# B&R Automation Studio project Panasonic_LinkaPowerCP2_A2021055 (part 7)

#### MaticaSet.st
```iecst
(* Skrutkovací set maticovačky *)
FUNCTION_BLOCK MaticaSet

	//Príznak matica pripravena//
	STAV.MaticaPripravena:= IN.PritomnostMaticeNaVystupe AND IN.PodavacMatice_ZASUNUTY;

	//*******************************Ovládanie zhadzovacieho vzduchu pred lištou zásobníka******************************************//
	Internal.CasZaplneniaZasobnika.IN:= IN.ZaplnenieListyZasobnika AND OUT.VibropohonZasobnika_RUN;

	IF Internal.CasZaplneniaZasobnika.Q THEN
		OUT.ZhadzovaciVzduch_RUN:= TRUE;
	ELSE
		OUT.ZhadzovaciVzduch_RUN:= FALSE;
	END_IF

	Internal.CasZaplneniaZasobnika.PT:= T#1s;
	Internal.CasZaplneniaZasobnika();

	//******************************Vypnutie triediaceho vzduchu nad lištou zásobníka************************************************//
	Internal.CasVypnTriediacehoVzduchu.IN:= OUT.TriediaciVzduch_RUN AND NOT OUT.VibropohonZasobnika_RUN;
	IF Internal.CasVypnTriediacehoVzduchu.Q THEN
		OUT.TriediaciVzduch_RUN:= FALSE;
	END_IF

	Internal.CasVypnTriediacehoVzduchu.PT:= T#1s;
	Internal.CasVypnTriediacehoVzduchu();

	//*******************************Vypnutie zásobníka***************************************//
	Internal.CasVypnZasobnika.IN:= IN.ZaplnenieListyZasobnika AND OUT.VibropohonZasobnika_RUN;

	IF Internal.CasVypnZasobnika.Q THEN
		OUT.VibropohonZasobnika_RUN:= FALSE;
	END_IF

	Internal.CasVypnZasobnika.PT:= T#3s;
	Internal.CasVypnZasobnika();

	//*******************************Zapnutie zásobníka keď je prázdna lišta zásobníka*****************//
	IF CMD.ENABLE AND NOT STAV.ERROR AND NOT IN.ZaplnenieListyZasobnika AND NOT OUT.VibropohonZasobnika_RUN AND IN.PodavacMatice_ZASUNUTY THEN
		OUT.VibropohonZasobnika_RUN:= TRUE;
	END_IF

	//***********************************Enable knižnice***************************************//
	IF NOT CMD.ENABLE AND Step <> 0 THEN
		OUT.VibropohonZasobnika_RUN:= FALSE;
		OUT.ZhadzovaciVzduch_RUN:= FALSE;
		OUT.NastrelenieMatice_RUN:= FALSE;
		Internal.PoInit:= FALSE;
		STAV.ERROR:= FALSE;
		STAV.PodanieMatice_BUSY:= FALSE;
		STAV.CisloPoruchy:= 0;
		STAV.PopisPoruchy:= '';
		Step:= 0;
	END_IF

	//**********************************Reset poruchy*****************************************//
	//1 - porucha preletu matice cez snímač za oddelovačom
	//2 - porucha preletu matice cez snimač pred podavačom
	//3 - porucha otočenia oddelovača smerom k zásobníku
	//4 - porucha otočenia oddelovača smerom k maticovačke
	//5 - porucha vysunutia podavača vpred
	//6 - porucha zasunutia podavača vzad
	//7 - porucha snimača prítomnosti matice v skrutkovačke

	IF CMD.ResetPoruchy THEN
		STAV.ERROR:= FALSE;
		STAV.CisloPoruchy:= 0;
		STAV.PopisPoruchy:= '';
	END_IF

	CASE Step OF

		0: //Nulovanie//
			Internal.IdleTime_200ms.IN:= FALSE;
			Internal.IdleTime_100ms.IN:= FALSE;
			Internal.IdleTime_500ms.IN:= FALSE;
			Internal.IdleTime_1s.IN:= FALSE;
			Internal.IdleTime_1500ms.IN:= FALSE;
			Internal.AlarmTime_3s.IN:= FALSE;
			OUT.PodavacMatice_Vysun:= FALSE;
			OUT.OtocOddelovacMatice_NaVystup:= FALSE;
			OUT.NastrelenieMatice_RUN:= FALSE;
			CMD.RR_OtocPodavac_Vstup:= FALSE;
			CMD.RR_OtocPodavac_Vystup:= FALSE;
			CMD.RR_VysunPodavacMatic:= FALSE;
			CMD.RR_ZapniZasobnik:= FALSE;
			CMD.RucnyRezim:= FALSE;
			CMD.PodajMaticu:=FALSE;
			STAV.PodanieMatice_BUSY:= FALSE;
			IF NOT CMD.PodajMaticu AND CMD.ENABLE AND NOT STAV.ERROR THEN
				Step:= 1;
			END_IF

		1: //Čakam na spustenie//
			IF CMD.RucnyRezim THEN
				Step:= 70;
			ELSIF CMD.PodajMaticu THEN
				Step:= 10;
			END_IF

		10: //Kontrola matice na vystupe//
			STAV.PodanieMatice_BUSY:= TRUE;
			IF IN.PritomnostMaticeNaVystupe THEN
				Step:= 0;
			ELSE
				IF NOT Internal.PoInit THEN
					Step:= 11;
				ELSE
					Step:= 13;
				END_IF
			END_IF

		11: //Hladanie matice pri prvom spusteni//
			OUT.PodavacMatice_Vysun:= FALSE;
			Internal.IdleTime_1500ms.IN:= OUT.NastrelenieMatice_RUN;

			IF IN.PodavacMatice_ZASUNUTY THEN
				OUT.NastrelenieMatice_RUN:= TRUE;
			END_IF

			IF Internal.IdleTime_1500ms.Q THEN
				OUT.NastrelenieMatice_RUN:= FALSE;
				Internal.IdleTime_1500ms.IN:= FALSE;
				Step:= 12;
			END_IF

		12: //Vysunutie podavača//
			OUT.PodavacMatice_Vysun:= TRUE;
			Internal.AlarmTime_3s.IN:= TRUE;
			Internal.IdleTime_500ms.IN:= IN.PodavacMatice_VYSUNUTY;

			IF Internal.IdleTime_500ms.Q THEN
				Internal.PoInit:= TRUE;
				Internal.IdleTime_500ms.IN:= FALSE;
				OUT.PodavacMatice_Vysun:= FALSE;
				Internal.AlarmTime_3s.IN:= FALSE;
				Step:= 10;
			ELSIF Internal.AlarmTime_3s.Q THEN
				STAV.ERROR:= TRUE;
				STAV.CisloPoruchy:= 5;
				STAV.PopisPoruchy:= 'Porucha vysunutia podavača vpred';
				Step:= 0;
			END_IF

		13: //Zasunutie podavaca matice a otocenie oddelovaca k zasobniku//
			OUT.PodavacMatice_Vysun:= FALSE;
			OUT.OtocOddelovacMatice_NaVystup:= FALSE;
			Internal.AlarmTime_3s.IN:= TRUE;

			IF IN.PodavacMatice_ZASUNUTY AND IN.OddelovacOtoceny_VSTUP THEN
				Internal.AlarmTime_3s.IN:= FALSE;
				Step:= 15;
			ELSIF Internal.AlarmTime_3s.Q THEN
				STAV.ERROR:= TRUE;
				IF NOT IN.PodavacMatice_ZASUNUTY THEN
					STAV.CisloPoruchy:= 6;
					STAV.PopisPoruchy:= 'Porucha zasunutia podavača vzad';
				ELSIF NOT IN.OddelovacOtoceny_VSTUP THEN
					STAV.CisloPoruchy:= 3;
					STAV.PopisPoruchy:= 'Porucha otocenia oddelovaca smerom k zasobníku';
				END_IF
				Step:= 0;
			END_IF

		15: //Spustenie zasobnika//
			OUT.TriediaciVzduch_RUN:= TRUE;
			Internal.IdleTime_1s.IN:= OUT.TriediaciVzduch_RUN;
			Internal.IdleTime_1500ms.IN:= IN.ZaplnenieListyZasobnika AND OUT.VibropohonZasobnika_RUN;

			IF Internal.IdleTime_1s.Q THEN
				OUT.VibropohonZasobnika_RUN:= TRUE;
			END_IF

			IF Internal.IdleTime_1500ms.Q THEN
				Internal.IdleTime_1s.IN:= FALSE;
				Internal.IdleTime_1500ms.IN:= FALSE;
				Step:= 18;
			END_IF

		18: //Otočenie oddelovača matic na vystup smerom k maticovačke a čakanie na prechod matice cez prvy snimac//
			OUT.OtocOddelovacMatice_NaVystup:= TRUE;
			Internal.AlarmTime_3s.IN:= TRUE;

			IF IN.Oddelovac_SnimPrechoduMatice THEN
				Internal.AlarmTime_3s.IN:= FALSE;
				Step:= 20;
			ELSIF Internal.AlarmTime_3s.Q THEN
				STAV.ERROR:= TRUE;
				STAV.CisloPoruchy:= 1;
				STAV.PopisPoruchy:= 'Porucha preletu matice cez snimac za oddelovacom';
				Step:= 0;
			END_IF

		20: //Zapnutie nastrelovacieho vzduchu a čakanie na prechod matice cez druhý snímač//
			OUT.NastrelenieMatice_RUN:= TRUE;
			Internal.AlarmTime_3s.IN:= TRUE;

			IF IN.Podavac_SnimPrechoduMatice THEN
				Internal.AlarmTime_3s.IN:= FALSE;
				Step:= 23;
			ELSIF Internal.AlarmTime_3s.Q THEN
				STAV.ERROR:= TRUE;
				STAV.CisloPoruchy:= 2;
				STAV.PopisPoruchy:= 'Porucha preletu matice cez snimac pred podavacom';
				Step:= 0;
			END_IF

		23: //Cakam na vysunutie podavaca//
			Internal.IdleTime_500ms.IN:= TRUE;

			IF Internal.IdleTime_500ms.Q THEN
				OUT.PodavacMatice_Vysun:= TRUE;
				Internal.AlarmTime_3s.IN:= TRUE;
			END_IF

			IF IN.PodavacMatice_VYSUNUTY AND IN.PritomnostMaticeNaVystupe THEN
				Internal.IdleTime_500ms.IN:= FALSE;
				Internal.AlarmTime_3s.IN:= FALSE;
				Step:= 25;
			ELSIF Internal.AlarmTime_3s.Q THEN
				STAV.ERROR:= TRUE;
				IF NOT IN.PodavacMatice_VYSUNUTY THEN
					STAV.CisloPoruchy:= 5;
					STAV.PopisPoruchy:= 'Porucha vysunutia podavaca vpred';
				ELSIF NOT IN.PritomnostMaticeNaVystupe THEN
					STAV.CisloPoruchy:= 7;
					STAV.PopisPoruchy:= 'Porucha snimaca pritomnosti matice v skrutkovacke';
				END_IF
				Step:= 0;
			END_IF

		25: //Čakam na zasunutie podavača//
			Internal.IdleTime_200ms.IN:= TRUE;

			IF Internal.IdleTime_200ms.Q THEN
				OUT.PodavacMatice_Vysun:= FALSE;
				Internal.AlarmTime_3s.IN:= TRUE;
			END_IF

			IF IN.PodavacMatice_ZASUNUTY THEN
				Internal.IdleTime_200ms.IN:= FALSE;
				Internal.AlarmTime_3s.IN:= FALSE;
				Step:= 0;
			ELSIF Internal.AlarmTime_3s.Q THEN
				STAV.ERROR:= TRUE;
				STAV.CisloPoruchy:= 6;
				STAV.PopisPoruchy:= 'Porucha zasunutia podavaca vzad';
				Step:= 0;
			END_IF

		70: //Rucny rezim//
			IF CMD.RR_ZapniZasobnik THEN
				OUT.TriediaciVzduch_RUN:= TRUE;
				Internal.IdleTime_1s.IN:= TRUE;
			ELSE
				Internal.IdleTime_1s.IN:= FALSE;
			END_IF

			OUT.VibropohonZasobnika_RUN:= Internal.IdleTime_1s.Q;

			IF NOT CMD.RucnyRezim THEN
				OUT.VibropohonZasobnika_RUN:= FALSE;
				Step:= 0;
			ELSIF CMD.PodajMaticu THEN
				OUT.PodavacMatice_Vysun:= FALSE;
				Step:= 10;
			END_IF

			IF CMD.RR_OtocPodavac_Vstup THEN
				OUT.OtocOddelovacMatice_NaVystup:= FALSE;
				CMD.RR_OtocPodavac_Vstup:= FALSE;
			ELSIF CMD.RR_OtocPodavac_Vystup THEN
				OUT.OtocOddelovacMatice_NaVystup:= TRUE;
				CMD.RR_OtocPodavac_Vystup:= FALSE;
			END_IF

			OUT.PodavacMatice_Vysun:= CMD.RR_VysunPodavacMatic;

	END_CASE

	//*****************Časovače************************//
	Internal.IdleTime_100ms.PT:= T#200ms;
	Internal.IdleTime_100ms();
	Internal.IdleTime_200ms.PT:= T#200ms;
	Internal.IdleTime_200ms();
	Internal.IdleTime_500ms.PT:= T#200ms;
	Internal.IdleTime_500ms();
	Internal.IdleTime_1s.PT:= T#1s;
	Internal.IdleTime_1s();
	Internal.IdleTime_1500ms.PT:= T#1s500ms;
	Internal.IdleTime_1500ms();
	Internal.AlarmTime_3s.PT:= T#40s;
	Internal.AlarmTime_3s();

END_FUNCTION_BLOCK
```

### Library Logical/Libraries/RoCa_Festo (IEC, version 1.00.0)

#### Types.typ - Exported data types
```iecst
TYPE
	OutputRawStruc : 	STRUCT
		Control_word_or_setpoint_0 : UINT;
		Control_word_or_setpoint_1 : UINT;
		Control_word_or_setpoint_2 : UINT;
		Control_word_or_setpoint_3 : UINT;
		Control_word_or_setpoint_4 : UINT;
		Control_word_or_setpoint_5 : UINT;
		Control_word_or_setpoint_6 : UINT;
		Control_word_or_setpoint_7 : UINT;
		Control_word_or_setpoint_8 : UINT;
		Control_word_or_setpoint_9 : UINT;
		Control_word_or_setpoint_10 : UINT;
		Control_word_or_setpoint_11 : UINT;
		Control_word_or_setpoint_12 : UINT;
		Control_word_or_setpoint_13 : UINT;
		Control_word_or_setpoint_14 : UINT;
		Control_word_or_setpoint_15 : UINT;
		User1 : UINT;
		MDI_decceleration : UINT;
		MDI_acceleration : UINT;
		MDI_velocity : UDINT;
		MDI_target_position : UDINT;
		Override : UINT;
		Position_Controlword_2 : UINT;
		Position_Controlword_1 : UINT;
		Control_word_2 : UINT;
		Control_word_1 : UINT;
	END_STRUCT;
	InputRawStruc : 	STRUCT
		Status_word_or_actual_value_0 : UINT;
		Status_word_or_actual_value_1 : UINT;
		Status_word_or_actual_value_2 : UINT;
		Status_word_or_actual_value_3 : UINT;
		Status_word_or_actual_value_4 : UINT;
		Status_word_or_actual_value_5 : UINT;
		Status_word_or_actual_value_6 : UINT;
		Status_word_or_actual_value_7 : UINT;
		Status_word_or_actual_value_8 : UINT;
		Status_word_or_actual_value_9 : UINT;
		Status_word_or_actual_value_10 : UINT;
		Status_word_or_actual_value_11 : UINT;
		Status_word_or_actual_value_12 : UINT;
		Status_word_or_actual_value_13 : UINT;
		Status_word_or_actual_value_14 : UINT;
		Status_word_or_actual_value_15 : UINT;
		User : UINT;
		Warn_Code : UINT;
		Fault_Code : UINT;
		Speed_actual_value_B : UDINT;
		Position_actual_value_A : UDINT;
		Report_word : UINT;
		Position_Statusword_2 : UINT;
		Position_Statusword_1 : UINT;
		Status_word_2 : UINT;
		Status_word_1 : UINT;
	END_STRUCT;
	OutputStruc : 	STRUCT
		ExtendedParam0 : UINT;
		ExtendedParam1 : UINT;
		ExtendedParam2 : UINT;
		ExtendedParam3 : UINT;
		ExtendedParam4 : UINT;
		ExtendedParam5 : UINT;
		ExtendedParam6 : UINT;
		ExtendedParam7 : UINT;
		ExtendedParam8 : UINT;
		ExtendedParam9 : UINT;
		ExtendedParam10 : UINT;
		ExtendedParam11 : UINT;
		ExtendedParam12 : UINT;
		ExtendedParam13 : UINT;
		ExtendedParam14 : UINT;
		ExtendedParam15 : UINT;
		user : UINT;
		TraverseToFixedEndstop_Bit8 : BOOL;
		ActivateHardwLimitSwitch_Bit15 : BOOL;
		ActivateSoftLimitSwitch_Bit14 : BOOL;
		TouchProbeEdgeSelection_Bit11 : BOOL;
		TouchProbeSelection_Bit10 : BOOL;
		JoggingIncremental_Bit5 : BOOL;
		MDIselection_Bit15 : BOOL;
		NegModuloPositioningDir_Bit10 : BOOL;
		PosModuloPositioningDir_Bit9 : BOOL;
		AbsolutePositioning_Bit8 : BOOL;
		TraversingBlockSelection_Bit0 : BOOL;
		TraversingBlockSelection_Bit1 : BOOL;
		TraversingBlockSelection_Bit2 : BOOL;
		TraversingBlockSelection_Bit3 : BOOL;
		TraversingBlockSelection_Bit4 : BOOL;
		TraversingBlockSelection_Bit5 : BOOL;
		TraversingBlockSelection_Bit6 : BOOL;
		OpenHoldingBrake_Bit12 : BOOL;
		StartHomingProcedure_Bit11 : BOOL;
		ControlByPLC_Bit10 : BOOL;
		Jog2_Bit9 : BOOL;
		Jog1_Bit8 : BOOL;
		FaultAck_Bit7 : BOOL;
		ActivateTraversingTask_Bit6 : BOOL;
		NoIntermediateStop_Bit5 : BOOL;
		DoNotRejectTraversingTask_Bit4 : BOOL;
		EnableOperation_Bit3 : BOOL;
		NoQuickStop_Bit2 : BOOL;
		NoCoastStop_Bit1 : BOOL;
		SwitchON_Bit0 : BOOL;
	END_STRUCT;
	InputStruc : 	STRUCT
		ExtendedParam0 : UINT;
		ExtendedParam1 : UINT;
		ExtendedParam2 : UINT;
		ExtendedParam3 : UINT;
		ExtendedParam4 : UINT;
		ExtendedParam5 : UINT;
		ExtendedParam6 : UINT;
		ExtendedParam7 : UINT;
		ExtendedParam8 : UINT;
		ExtendedParam9 : UINT;
		ExtendedParam10 : UINT;
		ExtendedParam11 : UINT;
		ExtendedParam12 : UINT;
		ExtendedParam13 : UINT;
		ExtendedParam14 : UINT;
		ExtendedParam15 : UINT;
		User : UINT;
		WarnCode : UINT;
		FaultCode : UINT;
		Speed : UDINT;
		Position : UDINT;
		PulsesEnabledMELDW_Bit13 : BOOL;
		DriveReady_Bit12 : BOOL;
		ControlerEnabled_Bit11 : BOOL;
		SpeedSetpointDeviationInTol_Bit8 : BOOL;
		PsTempWarningInactive_Bit7 : BOOL;
		MotorTempWarningInactive_Bit6 : BOOL;
		VariableSignalingFunction_Bit5 : BOOL;
		RPMequalThreshold_Bit3 : BOOL;
		RPMlowerThreshold_Bit2 : BOOL;
		TorqUtilLessTorqThres_Bit1 : BOOL;
		RampFunctionCompleted_Bit0 : BOOL;
		PulsesEnabled_Bit11 : BOOL;
		MoveToFixedStopActiveZSW2_Bit8 : BOOL;
		TraversingCommandActive_Bit15 : BOOL;
		MoveToFixedStopActive_Bit14 : BOOL;
		FixedStopClampTorqReached_Bit13 : BOOL;
		FixedStopReached_Bit12 : BOOL;
		DirectOut2ViaTraversBlock_Bit11 : BOOL;
		DirectOut1ViaTraversBlock_Bit10 : BOOL;
		PosActValueLessCamSwitch1_Bit9 : BOOL;
		PosActValueLessCamSwitch0_Bit8 : BOOL;
		SoftwareLimitSwitchPlus_Bit7 : BOOL;
		SoftwareLimitSwitchMinus_Bit6 : BOOL;
		DriveMovesBackwards_Bit5 : BOOL;
		DriveMovesForward_Bit4 : BOOL;
		SetpointAvailable_Bit2 : BOOL;
		VelocityLimitingActive_Bit1 : BOOL;
		TrackingModeActive_Bit0 : BOOL;
		MDIactive_Bit15 : BOOL;
		TraversingBlockActive_Bit13 : BOOL;
		RefPointAproachActive_Bit11 : BOOL;
		JoggingActive_Bit10 : BOOL;
		PositiveLimitSwitch_Bit9 : BOOL;
		NegativeLimitSwitch_Bit8 : BOOL;
		ActiveTravesringBlock_Bit0 : BOOL;
		ActiveTravesringBlock_Bit1 : BOOL;
		ActiveTravesringBlock_Bit2 : BOOL;
		ActiveTravesringBlock_Bit3 : BOOL;
		ActiveTravesringBlock_Bit4 : BOOL;
		ActiveTravesringBlock_Bit5 : BOOL;
		ActiveTravesringBlock_Bit6 : BOOL;
		AxisDeccelerated_Bit15 : BOOL;
		AxisAccelerated_Bit14 : BOOL;
		DriveStopped_Bit13 : BOOL;
		TraversingTaskAck_Bit12 : BOOL;
		HomePositionSet_Bit11 : BOOL;
		TargetPositionReached_Bit10 : BOOL;
		ControlRequested_Bit9 : BOOL;
		FolowingErrorWithinTol_Bit8 : BOOL;
		WarningPresent_Bit7 : BOOL;
		SwitchingOnInhibited_Bit6 : BOOL;
		QuickStopNotActivated_Bit5 : BOOL;
		CoastStopNotActivated_Bit4 : BOOL;
		FaultPresent_Bit3 : BOOL;
		OperationEnabled_Bit2 : BOOL;
		ReadyToOperate_Bit1 : BOOL;
		ReadyToSwitchON_Bit0 : BOOL;
	END_STRUCT;
	FestoServoDriverStruc : 	STRUCT
		OUT_forMapping : OutputRawStruc;
		IN_forMapping : InputRawStruc;
		OUT : OutputStruc;
		IN : InputStruc;
		Step : USINT;
		Info : WSTRING[80];
		Status : StatusStruc;
		Command : CommandStruc;
		Parameters : ParamStruc;
	END_STRUCT;
	ParamStruc : 	STRUCT
		Torque : REAL; (*Nm*)
		Distance : REAL; (*vzdialenost pre move additive [mm]*)
		Position : REAL; (*pozicia pre move position [mm]*)
		Override : REAL; (*0-200%*)
		Velocity : REAL; (*m/s*)
		Dcc : REAL; (*m/s2*)
		Acc : REAL; (*m/s2*)
		Jog : JogStruc;
	END_STRUCT;
	CommandStruc : 	STRUCT
		PowerON : BOOL;
		ErrReset : BOOL;
		JogNeg : BOOL;
		JogPos : BOOL;
		MoveAdditive : BOOL;
		MovePosition : BOOL;
		TorqueLimitation : BOOL; (*1-orezava moment na nastaveny v parametroch*)
		Stop : BOOL;
		Pause : BOOL;
	END_STRUCT;
	StatusStruc : 	STRUCT
		WarningMessage : WSTRING[80];
		ErrorMessage : WSTRING[80];
		InTorque : BOOL;
		InPosition : BOOL;
		StandStill : BOOL;
		Warning : BOOL;
		Error : BOOL;
		Ready : BOOL;
		ActTorque : REAL; (*Nm*)
		ActVelocity : REAL; (*mm/s*)
		ActPosition : REAL; (*mm*)
	END_STRUCT;
	JogStruc : 	STRUCT
		Acc : REAL;
		Velocity : REAL;
	END_STRUCT;
	LinearScaling_InternalStruc : 	STRUCT
		ScaleFactor : REAL;
		Offset : REAL;
	END_STRUCT;
	LinearScaling_SettingStruc : 	STRUCT
		InputLowerLimit : REAL; (*Minimum ktore vie vstup dosiahnut*)
		InputUpperLimit : REAL; (*Maximum ktore vie vstup dosiahnut*)
		OutputLowerLimit : REAL; (*Minimum ktore ma vystup ukazovat*)
		OutputUpperLimit : REAL; (*Maximum ktore ma vystup ukazovat*)
	END_STRUCT;
END_TYPE
```

#### RoCa_Festo.fun - Exported functions and function blocks
```iecst
{REDUND_OK} FUNCTION_BLOCK ServoDriver (*Riadenie festo driverov*) (*$GROUP=User,$CAT=Motion,$GROUPICON=User.png,$CATICON=User.png*)
	VAR_INPUT
		IN_forMapping : InputRawStruc;
		IN : InputStruc;
		Command : CommandStruc;
		Parameters : ParamStruc;
	END_VAR
	VAR_OUTPUT
		OUT_forMapping : OutputRawStruc;
		OUT : OutputStruc;
		Step : USINT;
		Info : WSTRING[80];
		Status : StatusStruc;
	END_VAR
	VAR
		TwoUINTtoREAL1 : twoUINTtoREAL;
		TwoUINTtoREAL2 : twoUINTtoREAL;
		TwoUINTtoREAL3 : twoUINTtoREAL;
		REALtoTwoUINT1 : REALtoTwoUINT;
		REALtoTwoUINT2 : REALtoTwoUINT;
		REALtoTwoUINT3 : REALtoTwoUINT;
		zzEdge00000 : {REDUND_UNREPLICABLE} BOOL;
		zzEdge00001 : {REDUND_UNREPLICABLE} BOOL;
		zzEdge00002 : {REDUND_UNREPLICABLE} BOOL;
		zzEdge00003 : {REDUND_UNREPLICABLE} BOOL;
		zzEdge00004 : {REDUND_UNREPLICABLE} BOOL;
		zzEdge00005 : BOOL;
	END_VAR
END_FUNCTION_BLOCK

{REDUND_OK} FUNCTION_BLOCK twoUINTtoREAL (*TODO: Add your comment here*) (*$GROUP=User,$CAT=Conversion,$GROUPICON=User.png,$CATICON=User.png*)
	VAR_INPUT
		IN1 : UINT; (*Vstupna premenna cislo 1*)
		IN2 : UINT; (*Vstupna premenna cislo 2*)
		order : BOOL; (*Poradie 0=IN1 first, 1=IN2 first*)
	END_VAR
	VAR_OUTPUT
		Out : REAL; (*Výstup vo formate REAL*)
	END_VAR
	VAR
		NxtADR : UDINT;
	END_VAR
END_FUNCTION_BLOCK

{REDUND_OK} FUNCTION_BLOCK REALtoTwoUINT (*TODO: Add your comment here*) (*$GROUP=User,$CAT=Conversion,$GROUPICON=User.png,$CATICON=User.png*)
	VAR_INPUT
		IN : REAL; (*Vstup vo formate REAL*)
		order : BOOL; (*poradie vystupov 0=OUT1 first, 1=OUT2first*)
	END_VAR
	VAR_OUTPUT
		OUT1 : UINT; (*Vystup vo formate UINT*)
		OUT2 : UINT; (*Vystup vo formate UINT*)
	END_VAR
	VAR
		NxtADR : UDINT;
	END_VAR
END_FUNCTION_BLOCK

{REDUND_OK} FUNCTION_BLOCK Linear_scaling (*Linearne skalovanie*) (*$GROUP=ROCA,$CAT=Mathematics,$GROUPICON=User.png,$CATICON=User.png*)
	VAR_INPUT
		Input : REAL; (*Vstup na preskalovanie*)
		Setting : LinearScaling_SettingStruc; (*Nastavenia*)
	END_VAR
	VAR_OUTPUT
		Output : REAL; (*Preskalovany vystup*)
		Info : STRING[80];
	END_VAR
	VAR
		Internal : LinearScaling_InternalStruc; (*Interne hodnoty pre prepocty*)
	END_VAR
END_FUNCTION_BLOCK
```

#### FestoDrivers.st
```iecst
(* Riadenie festo driverov *)
FUNCTION_BLOCK ServoDriver

	TwoUINTtoREAL1.order:=1;
	TwoUINTtoREAL2.order:=1;
	REALtoTwoUINT1.order:=1;
	REALtoTwoUINT2.order:=1;
	REALtoTwoUINT3.order:=1;

	TwoUINTtoREAL1;
	TwoUINTtoREAL2;
	REALtoTwoUINT1;
	REALtoTwoUINT2;
	REALtoTwoUINT3;

	TwoUINTtoREAL1.IN1:=IN_forMapping.Status_word_or_actual_value_0;
	TwoUINTtoREAL1.IN2:=IN_forMapping.Status_word_or_actual_value_1;

	TwoUINTtoREAL2.IN1:=IN_forMapping.Status_word_or_actual_value_2;
	TwoUINTtoREAL2.IN2:=IN_forMapping.Status_word_or_actual_value_3;

	OUT.ExtendedParam0:=REALtoTwoUINT1.OUT1;
	OUT.ExtendedParam1:=REALtoTwoUINT1.OUT2;

	OUT.ExtendedParam2:=REALtoTwoUINT2.OUT1;
	OUT.ExtendedParam3:=REALtoTwoUINT2.OUT2;

	OUT.ExtendedParam4:=REALtoTwoUINT3.OUT1;
	OUT.ExtendedParam5:=REALtoTwoUINT3.OUT2;

	//INPUTS
	//status word 1
	IN.ReadyToSwitchON_Bit0:=IN_forMapping.Status_word_1.0;
	IN.ReadyToOperate_Bit1:=IN_forMapping.Status_word_1.1;
	IN.OperationEnabled_Bit2:=IN_forMapping.Status_word_1.2;
	IN.FaultPresent_Bit3:=IN_forMapping.Status_word_1.3;
	IN.CoastStopNotActivated_Bit4:=IN_forMapping.Status_word_1.4;
	IN.QuickStopNotActivated_Bit5:=IN_forMapping.Status_word_1.5;
	IN.SwitchingOnInhibited_Bit6:=IN_forMapping.Status_word_1.6;
	IN.WarningPresent_Bit7:=IN_forMapping.Status_word_1.7;
	IN.FolowingErrorWithinTol_Bit8:=IN_forMapping.Status_word_1.8;
	IN.ControlRequested_Bit9:=IN_forMapping.Status_word_1.9;
	IN.TargetPositionReached_Bit10:=IN_forMapping.Status_word_1.10;
	IN.HomePositionSet_Bit11:=IN_forMapping.Status_word_1.11;
	IN.TraversingTaskAck_Bit12:=IN_forMapping.Status_word_1.12;
	IN.DriveStopped_Bit13:=IN_forMapping.Status_word_1.13;
	IN.AxisAccelerated_Bit14:=IN_forMapping.Status_word_1.14;
	IN.AxisDeccelerated_Bit15:=IN_forMapping.Status_word_1.15;

	//status word 2
	IN.MoveToFixedStopActiveZSW2_Bit8:=IN_forMapping.Status_word_2.8;
	IN.PulsesEnabled_Bit11:=IN_forMapping.Status_word_2.11;

	//position status word 1
	IN.ActiveTravesringBlock_Bit0:=IN_forMapping.Position_Statusword_1.0;
	IN.ActiveTravesringBlock_Bit1:=IN_forMapping.Position_Statusword_1.1;
	IN.ActiveTravesringBlock_Bit2:=IN_forMapping.Position_Statusword_1.2;
	IN.ActiveTravesringBlock_Bit3:=IN_forMapping.Position_Statusword_1.3;
	IN.ActiveTravesringBlock_Bit4:=IN_forMapping.Position_Statusword_1.4;
	IN.ActiveTravesringBlock_Bit5:=IN_forMapping.Position_Statusword_1.5;
	IN.ActiveTravesringBlock_Bit6:=IN_forMapping.Position_Statusword_1.6;

	IN.NegativeLimitSwitch_Bit8:=IN_forMapping.Position_Statusword_1.8;
	IN.PositiveLimitSwitch_Bit9:=IN_forMapping.Position_Statusword_1.9;
	IN.JoggingActive_Bit10:=IN_forMapping.Position_Statusword_1.10;
	IN.RefPointAproachActive_Bit11:=IN_forMapping.Position_Statusword_1.11;

	IN.TraversingBlockActive_Bit13:=IN_forMapping.Position_Statusword_1.13;
	IN.MDIactive_Bit15:=IN_forMapping.Position_Statusword_1.15;

	//position status word 2
	IN.TrackingModeActive_Bit0:=IN_forMapping.Position_Statusword_2.0;
	IN.VelocityLimitingActive_Bit1:=IN_forMapping.Position_Statusword_2.1;
	IN.SetpointAvailable_Bit2:=IN_forMapping.Position_Statusword_2.2;

	IN.DriveMovesForward_Bit4:=IN_forMapping.Position_Statusword_2.4;
	IN.DriveMovesBackwards_Bit5:=IN_forMapping.Position_Statusword_2.5;
	IN.SoftwareLimitSwitchMinus_Bit6:=IN_forMapping.Position_Statusword_2.6;
	IN.SoftwareLimitSwitchPlus_Bit7:=IN_forMapping.Position_Statusword_2.7;
	IN.PosActValueLessCamSwitch0_Bit8:=IN_forMapping.Position_Statusword_2.8;
	IN.PosActValueLessCamSwitch1_Bit9:=IN_forMapping.Position_Statusword_2.9;
	IN.DirectOut1ViaTraversBlock_Bit10:=IN_forMapping.Position_Statusword_2.10;
	IN.DirectOut2ViaTraversBlock_Bit11:=IN_forMapping.Position_Statusword_2.11;
	IN.FixedStopReached_Bit12:=IN_forMapping.Position_Statusword_2.12;
	IN.FixedStopClampTorqReached_Bit13:=IN_forMapping.Position_Statusword_2.13;
	IN.MoveToFixedStopActive_Bit14:=IN_forMapping.Position_Statusword_2.14;
	IN.TraversingCommandActive_Bit15:=IN_forMapping.Position_Statusword_2.15;

	//report word
	IN.RampFunctionCompleted_Bit0:=IN_forMapping.Report_word.0;
	IN.TorqUtilLessTorqThres_Bit1:=IN_forMapping.Report_word.1;
	IN.RPMlowerThreshold_Bit2:=IN_forMapping.Report_word.2;
	IN.RPMequalThreshold_Bit3:=IN_forMapping.Report_word.3;

	IN.VariableSignalingFunction_Bit5:=IN_forMapping.Report_word.5;
	IN.MotorTempWarningInactive_Bit6:=IN_forMapping.Report_word.6;
	IN.PsTempWarningInactive_Bit7:=IN_forMapping.Report_word.7;
	IN.SpeedSetpointDeviationInTol_Bit8:=IN_forMapping.Report_word.8;

	IN.ControlerEnabled_Bit11:=IN_forMapping.Report_word.11;
	IN.DriveReady_Bit12:=IN_forMapping.Report_word.12;
	IN.PulsesEnabledMELDW_Bit13:=IN_forMapping.Report_word.13;

	//not bool variables
	IN.FaultCode:=IN_forMapping.Fault_Code;
	IN.Position:=IN_forMapping.Position_actual_value_A;
	IN.Speed:=IN_forMapping.Speed_actual_value_B;
	IN.WarnCode:=IN_forMapping.Warn_Code;

	//extended proces variables
	IN.ExtendedParam0:=IN_forMapping.Status_word_or_actual_value_0;
	IN.ExtendedParam1:=IN_forMapping.Status_word_or_actual_value_1;
	IN.ExtendedParam2:=IN_forMapping.Status_word_or_actual_value_2;
	IN.ExtendedParam3:=IN_forMapping.Status_word_or_actual_value_3;
	IN.ExtendedParam4:=IN_forMapping.Status_word_or_actual_value_4;
	IN.ExtendedParam5:=IN_forMapping.Status_word_or_actual_value_5;
	IN.ExtendedParam6:=IN_forMapping.Status_word_or_actual_value_6;
	IN.ExtendedParam7:=IN_forMapping.Status_word_or_actual_value_7;
	IN.ExtendedParam8:=IN_forMapping.Status_word_or_actual_value_8;
	IN.ExtendedParam9:=IN_forMapping.Status_word_or_actual_value_9;
	IN.ExtendedParam10:=IN_forMapping.Status_word_or_actual_value_10;
	IN.ExtendedParam11:=IN_forMapping.Status_word_or_actual_value_11;
	IN.ExtendedParam12:=IN_forMapping.Status_word_or_actual_value_12;
	IN.ExtendedParam13:=IN_forMapping.Status_word_or_actual_value_13;
	IN.ExtendedParam14:=IN_forMapping.Status_word_or_actual_value_14;
	IN.ExtendedParam15:=IN_forMapping.Status_word_or_actual_value_15;

	//OUTPUTS
	//control word 1
	OUT_forMapping.Control_word_1.0:=OUT.SwitchON_Bit0;
	OUT_forMapping.Control_word_1.1:=OUT.NoCoastStop_Bit1;
	OUT_forMapping.Control_word_1.2:=OUT.NoQuickStop_Bit2;
	OUT_forMapping.Control_word_1.3:=OUT.EnableOperation_Bit3;
	OUT_forMapping.Control_word_1.4:=OUT.DoNotRejectTraversingTask_Bit4;
	OUT_forMapping.Control_word_1.5:=OUT.NoIntermediateStop_Bit5;
	OUT_forMapping.Control_word_1.6:=OUT.ActivateTraversingTask_Bit6;
	OUT_forMapping.Control_word_1.7:=OUT.FaultAck_Bit7;
	OUT_forMapping.Control_word_1.8:=OUT.Jog1_Bit8;
	OUT_forMapping.Control_word_1.9:=OUT.Jog2_Bit9;
	OUT_forMapping.Control_word_1.10:=OUT.ControlByPLC_Bit10;
	OUT_forMapping.Control_word_1.11:=OUT.StartHomingProcedure_Bit11;
	OUT_forMapping.Control_word_1.12:=OUT.OpenHoldingBrake_Bit12;

	//control word 2
	OUT_forMapping.Control_word_2.8:=OUT.TraverseToFixedEndstop_Bit8;

	//position control word 1
	OUT_forMapping.Position_Controlword_1.0:=OUT.TraversingBlockSelection_Bit0;
	OUT_forMapping.Position_Controlword_1.1:=OUT.TraversingBlockSelection_Bit1;
	OUT_forMapping.Position_Controlword_1.2:=OUT.TraversingBlockSelection_Bit2;
	OUT_forMapping.Position_Controlword_1.3:=OUT.TraversingBlockSelection_Bit3;
	OUT_forMapping.Position_Controlword_1.4:=OUT.TraversingBlockSelection_Bit4;
	OUT_forMapping.Position_Controlword_1.5:=OUT.TraversingBlockSelection_Bit5;
	OUT_forMapping.Position_Controlword_1.6:=OUT.TraversingBlockSelection_Bit6;

	OUT_forMapping.Position_Controlword_1.8:=OUT.AbsolutePositioning_Bit8;
	OUT_forMapping.Position_Controlword_1.9:=OUT.PosModuloPositioningDir_Bit9;
	OUT_forMapping.Position_Controlword_1.10:=OUT.NegModuloPositioningDir_Bit10;

	OUT_forMapping.Position_Controlword_1.15:=OUT.MDIselection_Bit15;

	//position control word 2
	OUT_forMapping.Position_Controlword_2.5:=OUT.JoggingIncremental_Bit5;

	OUT_forMapping.Position_Controlword_2.10:=OUT.TouchProbeSelection_Bit10;
	OUT_forMapping.Position_Controlword_2.11:=OUT.TouchProbeEdgeSelection_Bit11;

	OUT_forMapping.Position_Controlword_2.14:=OUT.ActivateSoftLimitSwitch_Bit14;
	OUT_forMapping.Position_Controlword_2.15:=OUT.ActivateHardwLimitSwitch_Bit15;

	//extended proces variables
	OUT_forMapping.Control_word_or_setpoint_0:=OUT.ExtendedParam0;
	OUT_forMapping.Control_word_or_setpoint_1:=OUT.ExtendedParam1;
	OUT_forMapping.Control_word_or_setpoint_2:=OUT.ExtendedParam2;
	OUT_forMapping.Control_word_or_setpoint_3:=OUT.ExtendedParam3;
	OUT_forMapping.Control_word_or_setpoint_4:=OUT.ExtendedParam4;
	OUT_forMapping.Control_word_or_setpoint_5:=OUT.ExtendedParam5;
	OUT_forMapping.Control_word_or_setpoint_6:=OUT.ExtendedParam6;
	OUT_forMapping.Control_word_or_setpoint_7:=OUT.ExtendedParam7;
	OUT_forMapping.Control_word_or_setpoint_8:=OUT.ExtendedParam8;
	OUT_forMapping.Control_word_or_setpoint_9:=OUT.ExtendedParam9;
	OUT_forMapping.Control_word_or_setpoint_10:=OUT.ExtendedParam10;
	OUT_forMapping.Control_word_or_setpoint_11:=OUT.ExtendedParam11;
	OUT_forMapping.Control_word_or_setpoint_12:=OUT.ExtendedParam12;
	OUT_forMapping.Control_word_or_setpoint_13:=OUT.ExtendedParam13;
	OUT_forMapping.Control_word_or_setpoint_14:=OUT.ExtendedParam14;
	OUT_forMapping.Control_word_or_setpoint_15:=OUT.ExtendedParam15;

	//prepocet aktualnych hodnot
	Status.ActPosition:=UDINT_TO_REAL (IN_forMapping.Position_actual_value_A)/100;
	Status.ActTorque:=TwoUINTtoREAL1.Out;
	Status.ActVelocity:=TwoUINTtoREAL2.Out;
	REALtoTwoUINT1.IN:=Parameters.Torque;
	REALtoTwoUINT2.IN:=Parameters.Jog.Velocity;
	REALtoTwoUINT3.IN:=Parameters.Jog.Acc;
	OUT_forMapping.Override:=REAL_TO_UINT(Parameters.Override*163.835);

	//switche
	OUT.TraverseToFixedEndstop_Bit8:=Command.TorqueLimitation;

	//statusy
	Status.InTorque:=IN.FixedStopClampTorqReached_Bit13;
	IF IN.DriveMovesBackwards_Bit5=0 AND IN.DriveMovesForward_Bit4=0 THEN Status.StandStill:=1; ELSE Status.StandStill:=0; END_IF

	//commandy
	//pauza
	IF Step>=100 THEN
		OUT.NoIntermediateStop_Bit5:=NOT (Command.Pause);
	END_IF
	//stop
	IF Step>=100 AND (IN.DriveMovesBackwards_Bit5=1 OR IN.DriveMovesForward_Bit4=1) THEN
		OUT.NoQuickStop_Bit2:=NOT (Command.Stop);
		IF EDGEPOS ( Command.Stop=1) THEN
			Step:=0;
		END_IF
	END_IF
	IF EDGENEG ( Command.Stop=1) THEN
		OUT.NoQuickStop_Bit2:=1;
		Step:=1;
	END_IF
	//PowerOFF
	IF Command.PowerON=0 THEN
		Step:=0;
	END_IF

	//Ready
	IF Step =100 OR Step=112 THEN
		IF IN.FaultPresent_Bit3=1 THEN Status.Ready:=0; ELSE Status.Ready:=1; END_IF
	ELSE
		Status.Ready:=0;
	END_IF

	//krokovy automat
	CASE Step OF
		0: Info:="Vypnute";
			OUT.AbsolutePositioning_Bit8:=0;
			OUT.ActivateHardwLimitSwitch_Bit15:=0;
			OUT.ActivateSoftLimitSwitch_Bit14:=0;
			OUT.ActivateTraversingTask_Bit6:=0;
			OUT.ControlByPLC_Bit10:=0;
			OUT.DoNotRejectTraversingTask_Bit4:=0;
			OUT.EnableOperation_Bit3:=0;
			OUT.FaultAck_Bit7:=0;
			OUT.Jog1_Bit8:=0;
			OUT.Jog2_Bit9:=0;
			OUT.JoggingIncremental_Bit5:=0;
			OUT.MDIselection_Bit15:=0;
			OUT.NegModuloPositioningDir_Bit10:=0;
			OUT.NoCoastStop_Bit1:=0;
			OUT.NoIntermediateStop_Bit5:=0;
			OUT.NoQuickStop_Bit2:=0;
			OUT.OpenHoldingBrake_Bit12:=0;
			OUT.PosModuloPositioningDir_Bit9:=0;
			OUT.StartHomingProcedure_Bit11:=0;
			OUT.SwitchON_Bit0:=0;
			OUT.TouchProbeEdgeSelection_Bit11:=0;
			OUT.TraverseToFixedEndstop_Bit8:=0;

			Status.Ready:=0;
			Status.InPosition:=0;

			IF Command.PowerON=1 THEN
				Step:=Step+1;
			END_IF

		1: Info:="Cakam na povolenie pristupu";
			OUT.ControlByPLC_Bit10:=1;
			IF IN.ControlRequested_Bit9=1 THEN
				Step:=Step+1;
			END_IF

		2: Info:="Cakam na zrusenie quick stop";
			OUT.NoIntermediateStop_Bit5:=1;
			OUT.NoQuickStop_Bit2:=1;
			IF IN.QuickStopNotActivated_Bit5=1 THEN
				Step:=Step+1;
			END_IF

		3: Info:="Cakam na zrusenie coast stop";
			OUT.NoCoastStop_Bit1:=1;
			IF IN.CoastStopNotActivated_Bit4=1 THEN
				Step:=Step+1;
			END_IF

		4: Info:="Cakam na zresetovanie chyby";
			Command.ErrReset:=1;
			IF IN.FaultCode=0 AND IN.WarnCode=0 THEN
				Command.ErrReset:=0;
				Step:=Step+1;
			END_IF

		5: Info:="rezerva";
			Step:=Step+1;

		6: Info:="Driver nie je pripraveny na spustenie";
			IF IN.ReadyToSwitchON_Bit0=1 THEN
				Step:=Step+1;
			END_IF

		7: Info:="Driver sa nepodarilo zapnut";
			OUT.SwitchON_Bit0:=1;
			IF IN.ReadyToOperate_Bit1=1 THEN
				Step:=Step+1;
			END_IF

		8: Info:="Vykonovu cast sa nepodarilo zapnut";
			OUT.EnableOperation_Bit3:=1;
			IF IN.OperationEnabled_Bit2=1 THEN
				Step:=Step+1;
			END_IF

		9: Info:="Nepodarilo sa aktivovat MDI";
			OUT.DoNotRejectTraversingTask_Bit4:=1;
			OUT.MDIselection_Bit15:=1;
			IF IN.MDIactive_Bit15=1 THEN
				Step:=Step+1;
			END_IF

		10:Step:=90;

		90: Info:="Cakam na zrusenie prikazu MOVE POSITION";
			IF Command.MovePosition=0 THEN
				Step:=Step+1;
			END_IF

		91: Info:="Cakam na zrusenie prikazu MOVE ADITIVE";
			IF Command.MoveAdditive=0 THEN
				Step:=Step+1;
			END_IF

		92: Info:="Cakam na zrusenie prikazu JOG POSITIVE";
			IF Command.JogPos=0 THEN
				Step:=Step+1;
			END_IF

		93: Info:="Cakam na zrusenie prikazu JOG NEGATIVE";
			IF Command.JogNeg=0 THEN
				Step:=Step+1;
			END_IF

		94:Step:=Step+1;
		95:Step:=Step+1;
		96:Step:=Step+1;
		97:Step:=Step+1;
		98:Step:=Step+1;
		99:Step:=Step+1;

		100:Info:="Pripraveny cakam na povel";

			OUT_forMapping.MDI_acceleration:=REAL_TO_UINT(Parameters.Acc*163.839989933671);
			OUT_forMapping.MDI_decceleration:=REAL_TO_UINT(Parameters.Dcc*163.839989933671);
			OUT_forMapping.MDI_velocity:=REAL_TO_UDINT(Parameters.Velocity*1000);
			OUT.ActivateSoftLimitSwitch_Bit14:=1;

			IF Command.MovePosition=1 AND IN.TraversingTaskAck_Bit12=0 THEN
				OUT.AbsolutePositioning_Bit8:=1;
				OUT_forMapping.MDI_target_position:=REAL_TO_UDINT(Parameters.Position*100);
				IF (Parameters.Position>=Status.ActPosition-0.05) AND (Parameters.Position<=Status.ActPosition+0.05) THEN
					Step:=113;
				ELSE
					Step:=110;
				END_IF
			ELSIF Command.MoveAdditive=1 THEN
				OUT.AbsolutePositioning_Bit8:=0;
				OUT_forMapping.MDI_target_position:=REAL_TO_UDINT(Parameters.Distance*100);
				Step:=120;
			ELSIF Command.JogPos=1 THEN
				Step:=130;
			ELSIF Command.JogNeg=1 THEN
				Step:=140;
			END_IF

			// move position
		110:Info:="Cakam na potvrdenie pohyboveho prikazu";
			OUT.ActivateTraversingTask_Bit6:=1;
			IF IN.TraversingTaskAck_Bit12=1 THEN
				Step:=Step+1;
			END_IF

		111:Info:="Cakam na potvrdenie pohyboveho prikazu";
			IF IN.TraversingCommandActive_Bit15=1 THEN
				Step:=Step+1;
			END_IF

		112:Info:="Cakam kym servo napolohuje";
			IF EDGEPOS (IN.TargetPositionReached_Bit10=1) THEN
				OUT.ActivateTraversingTask_Bit6:=0;
				Step:=Step+1;
			ELSIF EDGEPOS (Command.MovePosition=1) THEN
				OUT.ActivateTraversingTask_Bit6:=0;
				Step:=114;
			END_IF

		113:Info:="Cakam na zrusenie poziadavky na polohovanie";
			Status.InPosition:=1;
			IF Command.MovePosition=0 THEN
				Status.InPosition:=0;
				Step:=199;
			END_IF

		114:Info:="Cakam kym servo prerusi ulohu";
			IF IN.TraversingTaskAck_Bit12=0 THEN
				Step:=199;
			END_IF

			// move addition
		120:Info:="Cakam na potvrdenie pohyboveho prikazu";
			OUT.ActivateTraversingTask_Bit6:=1;
			IF IN.TraversingTaskAck_Bit12=1 THEN
				Step:=Step+1;
			END_IF

		121:Info:="Cakam kym servo napolohuje";
			IF IN.TargetPositionReached_Bit10=1 THEN
				OUT.ActivateTraversingTask_Bit6:=0;
				Step:=Step+1;
			END_IF

		122:Info:="Cakam na zrusenie poziadavky na polohovanie";
			Status.InPosition:=1;
			IF Command.MoveAdditive=0 THEN
				Status.InPosition:=0;
				Step:=199;
			END_IF
			// jog positive
		130:Info:="Jog positivnym smerom";
			IF Command.JogPos=1 THEN
				OUT.Jog1_Bit8:=1;
			ELSE
				OUT.Jog1_Bit8:=0;
				Step:=199;
			END_IF

		140:Info:="Jog negativnym smerom";
			IF Command.JogNeg=1 THEN
				OUT.Jog2_Bit9:=1;
			ELSE
				OUT.Jog2_Bit9:=0;
				Step:=199;
			END_IF
		199:
			Step:=100;
	END_CASE

	// chybove hlasky
	IF IN_forMapping.Fault_Code<>0 THEN
		Status.Error:=1;
	ELSE
		Status.Error:=0;
	END_IF
	CASE IN_forMapping.Fault_Code OF
		0: Status.ErrorMessage:="No error";
		36: Status.ErrorMessage:="Napajacie napatie nepritomne";
		38: Status.ErrorMessage:="Podpatie na napajani";
		73: Status.ErrorMessage:="Nespravna hodnota rychlosti/akceleracie";
		74: Status.ErrorMessage:="Nespravna hodnota akceleracie/deceleracie";
		109: Status.ErrorMessage:="Negativny softwareovy limit prekroceny";
		110: Status.ErrorMessage:="Pozitivny softwareovy limit prekroceny";
		141: Status.ErrorMessage:="Nespravne procesne data (velocity, override, acc, dcc...";

		ELSE
			Status.ErrorMessage:="Neznama chyba";
	END_CASE

	// varovania
	IF IN_forMapping.Warn_Code<>0 THEN
		Status.Warning:=1;
	ELSE
		Status.Warning:=0;
	END_IF
	CASE IN_forMapping.Warn_Code OF
		0: Status.WarningMessage:="No warning";
		37: Status.WarningMessage:="Prerusenie napajania";
		111: Status.WarningMessage:="Limit v negativnom smere";
		112: Status.WarningMessage:="Limit v pozitivnom smere";
		129: Status.WarningMessage:="Out of target range";
		364: Status.WarningMessage:="Nastavena rychlost = 0";

		ELSE
			Status.WarningMessage:="Nezname varovanie";
	END_CASE

	//reset poruch a varovani
	OUT.FaultAck_Bit7:=Command.ErrReset;
	IF Step>=100 AND IN.FaultPresent_Bit3=1 THEN
		IF EDGEPOS ( Command.ErrReset=1) THEN
			Step:=0;
		END_IF
	END_IF
	IF EDGENEG ( Command.ErrReset=1) THEN
		Step:=1;
	END_IF

END_FUNCTION_BLOCK
```

#### twoUINTtoREAL.st
```iecst
(* Poskladanie REAL z dvoch UINT *)
FUNCTION_BLOCK twoUINTtoREAL
	IF order = 0 THEN
		NxtADR := brsmemcpy(ADR(Out),ADR(IN1),2);
		NxtADR := brsmemcpy(ADR(Out)+2,ADR(IN2),2);
	ELSE
		NxtADR := brsmemcpy(ADR(Out),ADR(IN2),2);
		NxtADR := brsmemcpy(ADR(Out)+2,ADR(IN1),2);
	END_IF

END_FUNCTION_BLOCK
```

#### REALtoTwoUINT.st
```iecst
(* adresne rozobratie REAL do dvoch UINT (nie matematicky) *)
FUNCTION_BLOCK REALtoTwoUINT
	IF order=0 THEN
		NxtADR := brsmemcpy(ADR(OUT1),ADR(IN),2);
		NxtADR := brsmemcpy(ADR(OUT2),ADR(IN)+2,2);
	ELSE
		NxtADR := brsmemcpy(ADR(OUT1),ADR(IN)+2,2);
		NxtADR := brsmemcpy(ADR(OUT2),ADR(IN),2);
	END_IF

END_FUNCTION_BLOCK
```

#### Linear_scaling.st
```iecst
(* Linearne skalovanie verzia 1.0 *)
(* Powered by ROCA systems, s.r.o. *)
FUNCTION_BLOCK Linear_scaling
	//osetrenie delenia nulov
	IF Setting.InputUpperLimit-Setting.InputLowerLimit <> 0 THEN
		Internal.ScaleFactor:=(Setting.OutputUpperLimit-Setting.OutputLowerLimit)/(Setting.InputUpperLimit-Setting.InputLowerLimit);
	END_IF
	//vypocet offsetu
	Internal.Offset:=Setting.OutputLowerLimit-Internal.ScaleFactor*Setting.InputLowerLimit;
	//vypocet vystupu
	Output:=(Internal.ScaleFactor*Input)+Internal.Offset;

	//osetrenie hlasok
	IF Setting.InputUpperLimit-Setting.InputLowerLimit = 0 THEN Info:='Horny a dolny limit vstupu je rovnaky';
	ELSIF Setting.OutputUpperLimit-Setting.OutputLowerLimit = 0 THEN Info:='Horny a dolny limit vystupu je rovnaky';
	ELSIF Input<Setting.InputLowerLimit THEN Info:='Vstup je mensi ako zadany dolny limit vstupu';
	ELSIF Input>Setting.InputUpperLimit THEN Info:='Vstup je vacsi ako zadany horny limit vstupu';
	ELSE Info:='OK';
	END_IF

END_FUNCTION_BLOCK
```

### Library Logical/Libraries/Statistika (IEC)

#### Types.typ - Exported data types
```iecst
TYPE
	Statistika_IN_typ : 	STRUCT
		START_MeraniaCasu : BOOL;
		START_MeraniaStratovehoCasu : BOOL;
		ZAPIS_MeraniaCasu : BOOL;
		ZAPIS_StratovyCas : BOOL;
		TaskovaTrieda_ms : UINT;
		RESET_CelkovehoCasu : BOOL;
		RESET_HistorieMeraniCasu : BOOL;
		RESET_PoctuKusov : BOOL;
		RESET_CelkovehoPoctuKusov : BOOL;
		RESET_StratovehoCasu : BOOL;
		PriratajKus_OK : BOOL;
		PriratajKus_NG : BOOL;
	END_STRUCT;
	Statistika_OUT_typ : 	STRUCT
		NameranyCas_v_Sekundach : REAL;
		NameranyCas_v_Minutach : REAL;
		NameranyCas_v_Hodinach : REAL;
		PriemernyCas_v_Sekundach : REAL;
		PriemernyCas_v_Minutach : REAL;
		StratoveSekundy : REAL;
		StratoveMinuty : REAL;
		StratoveHodiny : REAL;
		HistoriaMerani_v_Sekundach : ARRAY[0..14]OF REAL;
		HistoriaMerani_v_Minutach : ARRAY[0..14]OF REAL;
		HistoriaMerani_v_Hodinach : ARRAY[0..14]OF REAL;
		CelkovyPocetNameranychSekund : REAL;
		CelkovyPocetNameranychMinut : REAL;
		CelkovyPocetNameranychHodin : REAL;
		PocetKusov_OK : UDINT;
		PocetKusov_NG : UDINT;
		CelkovyPocetKusov : UDINT;
	END_STRUCT;
	Statistika_VAR_typ : 	STRUCT
		NameraneMilisekundy_REAL : REAL;
		NameraneSekundy_REAL : REAL;
		NameraneMinuty_REAL : REAL;
		NameraneHodiny_REAL : REAL;
		Milisekundy : UINT;
		Sekundy : UINT;
		Minuty : UINT;
		Hodiny : UINT;
		CelkoveSekundy : UINT;
		CelkoveMinuty : UINT;
		CelkoveHodiny : UINT;
		i : USINT;
		a : USINT;
		b : USINT;
		c : USINT;
		d : USINT;
		Priemer_SucetSekund_REAL : REAL;
		Priemer_SucetMinut_REAL : REAL;
		Priemer_SucetHodin_REAL : REAL;
		StratoveMilisekundy : UINT;
		StratoveSekundy : UINT;
		StratoveMinuty : UINT;
		StratoveHodiny : UINT;
		CelkoveStratoveMilisekundy_REAL : REAL;
		CelkoveStratoveSekundy_REAL : REAL;
	END_STRUCT;
END_TYPE
```

#### Statistika.fun - Exported functions and function blocks
```iecst
{REDUND_ERROR} FUNCTION_BLOCK Taktime (*Meranie taktime*) (*$GROUP=User,$CAT=User,$GROUPICON=User.png,$CATICON=User.png*)
	VAR_INPUT
		IN : Statistika_IN_typ;
	END_VAR
	VAR_OUTPUT
		OUT : Statistika_OUT_typ;
	END_VAR
	VAR
		IntVAR : Statistika_VAR_typ;
	END_VAR
END_FUNCTION_BLOCK
```

#### Taktime.st
```iecst
(* Meranie taktime *)
FUNCTION_BLOCK Taktime

//*********************************************************************Meranie taktime**************************************************************************//

    //Vynulovanie časovača//
	IF NOT IN.START_MeraniaCasu THEN
		IntVAR.Milisekundy:= 0;
		IntVAR.Sekundy:= 0;
		IntVAR.Minuty:= 0;
		IntVAR.Hodiny:= 0;
		IntVAR.CelkoveSekundy:= 0;
		IntVAR.CelkoveMinuty:= 0;
		IntVAR.CelkoveHodiny:= 0;
		IntVAR.NameraneSekundy_REAL:= 0;
	END_IF

	//Zapnutie časovača//
	IF IN.START_MeraniaCasu THEN

		IntVAR.Milisekundy:= IntVAR.Milisekundy + IN.TaskovaTrieda_ms;//Ak je v taskovej triede 2ms tak prirátaváme + 2//

		IF IntVAR.Milisekundy >= 1000 THEN
			IntVAR.Sekundy:= IntVAR.Sekundy + 1;
			IntVAR.NameraneSekundy_REAL:= IntVAR.NameraneSekundy_REAL + 1;
			IntVAR.Milisekundy:= 0;
		END_IF

		IF IntVAR.Sekundy >= 60 THEN
			IntVAR.Minuty:= IntVAR.Minuty + 1;
			IntVAR.Sekundy:= 0;
		END_IF

		IF IntVAR.Minuty >= 60 THEN
			IntVAR.Hodiny:= IntVAR.Hodiny + 1;
			IntVAR.Minuty:= 0;
		END_IF

	END_IF

	//Ulozenie nameraného času a resetovanie časovača//
	IF IN.ZAPIS_MeraniaCasu THEN
		IntVAR.NameraneMilisekundy_REAL:= UINT_TO_REAL(IntVAR.Milisekundy);
		//Zobrazenie celkového času v sekundách//
		OUT.NameranyCas_v_Sekundach:= IntVAR.NameraneSekundy_REAL + (IntVAR.NameraneMilisekundy_REAL / 1000);
		//Zobrazenie celkového času v minútach//
		OUT.NameranyCas_v_Minutach:= OUT.NameranyCas_v_Sekundach / 60;
		//Zobrazenie celkového času v hodinách//
		OUT.NameranyCas_v_Hodinach:= OUT.NameranyCas_v_Minutach / 60;
		//Zápis do historie meraní//
		OUT.HistoriaMerani_v_Sekundach[IntVAR.i]:= OUT.NameranyCas_v_Sekundach;
		OUT.HistoriaMerani_v_Minutach[IntVAR.i]:= OUT.NameranyCas_v_Minutach;
		IntVAR.i:= IntVAR.i + 1;
		IF IntVAR.i > 14 THEN
			IntVAR.i:= 0;
		END_IF
		OUT.CelkovyPocetNameranychSekund:= OUT.CelkovyPocetNameranychSekund + OUT.NameranyCas_v_Sekundach;
		OUT.CelkovyPocetNameranychMinut:= OUT.CelkovyPocetNameranychMinut + OUT.NameranyCas_v_Minutach;
		OUT.CelkovyPocetNameranychHodin:= OUT.CelkovyPocetNameranychHodin + OUT.NameranyCas_v_Hodinach;
		IntVAR.Milisekundy:= 0;
		IntVAR.Sekundy:= 0;
		IntVAR.Minuty:= 0;
		IntVAR.Hodiny:= 0;
		IntVAR.CelkoveSekundy:= 0;
		IntVAR.CelkoveMinuty:= 0;
		IntVAR.CelkoveHodiny:= 0;
		IntVAR.NameraneSekundy_REAL:= 0;
		IN.ZAPIS_MeraniaCasu:= FALSE;
	END_IF

	//Vyrátanie priemernej hodnoty v sekundách//
	IntVAR.a:= 0;
	IntVAR.b:= 0;
	IntVAR.Priemer_SucetSekund_REAL:= 0;
	OUT.PriemernyCas_v_Sekundach:= 0;
	FOR IntVAR.a:= 0 TO 14 BY 1 DO
		IntVAR.Priemer_SucetSekund_REAL:= IntVAR.Priemer_SucetSekund_REAL + OUT.HistoriaMerani_v_Sekundach[IntVAR.a];
		IF OUT.HistoriaMerani_v_Sekundach[IntVAR.a] <> 0 THEN
			IntVAR.b:= IntVAR.b + 1;
		END_IF
		IF IntVAR.b <> 0 THEN
			OUT.PriemernyCas_v_Sekundach:= IntVAR.Priemer_SucetSekund_REAL / IntVAR.b;
		ELSE
			OUT.PriemernyCas_v_Sekundach:= 0;
		END_IF
	END_FOR

	//Vyrátanie priemernej hodnoty v minutách//
	IntVAR.c:= 0;
	IntVAR.d:= 0;
	IntVAR.Priemer_SucetMinut_REAL:= 0;
	OUT.PriemernyCas_v_Minutach:= 0;
	FOR IntVAR.c:= 0 TO 14 BY 1 DO
		IntVAR.Priemer_SucetMinut_REAL:= IntVAR.Priemer_SucetMinut_REAL + OUT.HistoriaMerani_v_Minutach[IntVAR.c];
		IF OUT.HistoriaMerani_v_Minutach[IntVAR.c] <> 0 THEN
			IntVAR.d:= IntVAR.d + 1;
		END_IF
		IF IntVAR.d <> 0 THEN
			OUT.PriemernyCas_v_Minutach:= IntVAR.Priemer_SucetMinut_REAL / IntVAR.d;
		ELSE
			OUT.PriemernyCas_v_Minutach:= 0;
		END_IF
	END_FOR

	//Reset celkových počítadiel času//
	IF IN.RESET_CelkovehoCasu THEN
		OUT.CelkovyPocetNameranychSekund:= 0;
		OUT.CelkovyPocetNameranychMinut:= 0;
		OUT.CelkovyPocetNameranychHodin:= 0;
		IN.RESET_CelkovehoCasu:= FALSE;
	END_IF

	//Reset historie merani//
	IF IN.RESET_HistorieMeraniCasu THEN
		brsmemset(ADR(OUT.HistoriaMerani_v_Sekundach),0,SIZEOF(OUT.HistoriaMerani_v_Sekundach));
		brsmemset(ADR(OUT.HistoriaMerani_v_Minutach),0,SIZEOF(OUT.HistoriaMerani_v_Minutach));
		IN.RESET_HistorieMeraniCasu:= FALSE;
	END_IF

	//***************************************************************************Rátanie kusov****************************************************************************//

	//Rátanie kusov OK//
	IF IN.PriratajKus_OK THEN
		OUT.CelkovyPocetKusov:= OUT.CelkovyPocetKusov + 1;
		OUT.PocetKusov_OK:= OUT.PocetKusov_OK + 1;
		IN.PriratajKus_OK:= FALSE;
	END_IF

	//Rátanie kusov NG//
	IF IN.PriratajKus_NG THEN
		OUT.CelkovyPocetKusov:= OUT.CelkovyPocetKusov + 1;
		OUT.PocetKusov_NG:= OUT.PocetKusov_NG + 1;
		IN.PriratajKus_NG:= FALSE;
	END_IF

	//Reset počtu kusov //
	IF IN.RESET_PoctuKusov THEN
		OUT.PocetKusov_OK:= 0;
		OUT.PocetKusov_NG:= 0;
		IN.RESET_PoctuKusov:= FALSE;
	END_IF

	//Reset celkového počtu kusov//
	IF IN.RESET_CelkovehoPoctuKusov THEN
		OUT.CelkovyPocetKusov:= 0;
		IN.RESET_CelkovehoPoctuKusov:= FALSE;
	END_IF

  //*********************************************Meranie stratoveho času*****************************************//

	//Spustenie merania//
	IF IN.START_MeraniaStratovehoCasu THEN

		IntVAR.StratoveMilisekundy:= IntVAR.StratoveMilisekundy + IN.TaskovaTrieda_ms;//Ak je v taskovej triede 2ms tak prirátaváme + 2//

		IF IntVAR.StratoveMilisekundy >= 1000 THEN
			IntVAR.StratoveSekundy:= IntVAR.StratoveSekundy + 1;
			IntVAR.CelkoveStratoveSekundy_REAL:= IntVAR.CelkoveStratoveSekundy_REAL + 1;
			IntVAR.StratoveMilisekundy:= 0;
		END_IF

		IF IntVAR.StratoveSekundy >= 60 THEN
			IntVAR.StratoveMinuty:= IntVAR.StratoveMinuty + 1;
			IntVAR.StratoveSekundy:= 0;
		END_IF

		IF IntVAR.StratoveMinuty >= 60 THEN
			IntVAR.StratoveHodiny:= IntVAR.StratoveHodiny + 1;
			IntVAR.StratoveMinuty:= 0;
		END_IF

	END_IF

	//Zapísanie stratového času//
	IF IN.ZAPIS_StratovyCas THEN
		//Zobrazenie celkového času v sekundách//
		IntVAR.CelkoveStratoveMilisekundy_REAL:= UINT_TO_REAL(IntVAR.StratoveMilisekundy);
		OUT.StratoveSekundy:= IntVAR.CelkoveStratoveSekundy_REAL + (IntVAR.CelkoveStratoveMilisekundy_REAL / 1000);
		//Zobrazenie celkového času v minútach//
		OUT.StratoveMinuty:= OUT.StratoveSekundy / 60;
		//Zobrazenie celkového času v hodinách//
		OUT.StratoveHodiny:= OUT.StratoveMinuty / 60;
		IntVAR.StratoveMilisekundy:= 0;
		IntVAR.CelkoveStratoveSekundy_REAL:= 0;
		IN.ZAPIS_StratovyCas:= FALSE;
	END_IF

	//Reset merania//

	IF IN.RESET_StratovehoCasu THEN
		IntVAR.StratoveMilisekundy:= 0;
		IntVAR.CelkoveStratoveSekundy_REAL:= 0;
		OUT.StratoveSekundy:= 0;
		IN.RESET_StratovehoCasu:= FALSE;
	END_IF

END_FUNCTION_BLOCK
```

### Library Logical/Libraries/ScrewLoad (IEC, version 1.00.0)

#### Types.typ - Exported data types
```iecst
(*--- Vibracny hrniec ---*)

TYPE
	VibracnyHrniecStruc : 	STRUCT
		IN : VibracnyHrniecIN;
		OUT : VibracnyHrniecOUT;
		Premenne : VibracnyHrniecVAR;
	END_STRUCT;
	VibracnyHrniecIN : 	STRUCT
		PritomnostSkrutiekVHrnci : BOOL;
		VibracnaListaZaplnena : BOOL;
		PreletovySnimac : BOOL;
	END_STRUCT;
	VibracnyHrniecOUT : 	STRUCT
		PrerusenieZasobovaniaSkrutiek : BOOL;
		TiedenieSkrutiek : BOOL;
		VzduchNastreleniaSkrutky : BOOL;
		OddelovacVysunut : BOOL;
		ZapniVibromotor : BOOL;
	END_STRUCT;
	VibracnyHrniecVAR : 	STRUCT
		T_ZapnutieTriediacehoVzduchu : TON;
		T_Zaplnenie : TON;
		T_PreletSkrutky : TON;
		T_PredOpatovnymPodanimSkrutky : TON;
	END_STRUCT;
END_TYPE

(*--- Brzda ---*)

TYPE
	BrzdaStruc : 	STRUCT
		IN : BrzdaIN;
		OUT : BrzdaOUT;
		Premenne : BrzdaVAR;
	END_STRUCT;
	BrzdaIN : 	STRUCT
		ZakladnaPoloha : BOOL;
		PodajSkrutku : BOOL;
		PreletSkrutky : BOOL;
		SkrutkaPritomnaVBrzde : BOOL;
		VyziadanieSkrutky : BOOL;
	END_STRUCT;
	BrzdaOUT : 	STRUCT
		ZakladnaPoloha : BOOL;
		PodajSkrutku : BOOL;
		OdsavanieNecistot : BOOL;
		SktutkaPodana : BOOL;
		NastrelenieSkrutky : BOOL;
	END_STRUCT;
	BrzdaVAR : 	STRUCT
		T_PreletSkrutky : TON;
		T_CasCisteniaSkrutky : TON;
		T_PresunBrzdy : TON;
	END_STRUCT;
END_TYPE

(*--- Brzda ---*)

TYPE
	StepStruc_typ : 	STRUCT
		VibracnyHrniec : USINT;
		Brzda : USINT;
	END_STRUCT;
	StatusStruc_typ : 	STRUCT
		VibracnyHrniec : WSTRING[80];
		Brzda : WSTRING[80];
	END_STRUCT;
END_TYPE

(*--- Struktura ---*)

TYPE
	InternalStruc : 	STRUCT
		Brzda : BrzdaVAR;
		VibracnyHrniec : VibracnyHrniecVAR;
		Step : StepStruc_typ;
		Status : StatusStruc_typ;
	END_STRUCT;
	ErrorStruc_typ : 	STRUCT
		ErrorBit : BOOL;
		ErrorNumber : UINT;
		ErrorMessage : WSTRING[80];
	END_STRUCT;
	StatusFBStruc : 	STRUCT
		AutomatBezi : BOOL;
		ManualBeziHrniec : BOOL;
		SkrutkaPripravena : BOOL;
	END_STRUCT;
	CmdStruc : 	STRUCT
		AutomatStart : BOOL;
		ManualPresunBrzdu : BOOL;
		ManualStartHrniec : BOOL;
		PodajSkrutku : BOOL;
	END_STRUCT;
	OutStruc : 	STRUCT
		Brzda : BrzdaOUT;
		VibracnyHrniec : VibracnyHrniecOUT;
	END_STRUCT;
	InStruc : 	STRUCT
		Brzda : BrzdaIN;
		VibracnyHrniec : VibracnyHrniecIN;
	END_STRUCT;
END_TYPE
```

#### ScrewLoad.fun - Exported functions and function blocks
```iecst
{REDUND_ERROR} FUNCTION_BLOCK ScrewLoading (*Nabíjanie skrutiek pre systém WEBER*) (*$GROUP=User,$CAT=User,$GROUPICON=User.png,$CATICON=User.png*)
	VAR_INPUT
		Cmd : {REDUND_UNREPLICABLE} CmdStruc; (*Ovládacie príkazy*)
		IN : InStruc;
	END_VAR
	VAR_OUTPUT
		Status : StatusFBStruc; (*Statusové bity*)
		Error : {REDUND_UNREPLICABLE} ErrorStruc_typ; (*Chybové hlásenia*)
		OUT : OutStruc;
	END_VAR
	VAR
		Internal : InternalStruc;
		zzEdge00000 : BOOL;
		zzEdge00001 : BOOL;
		zzEdge00002 : BOOL;
		zzEdge00003 : BOOL;
		zzEdge00004 : BOOL;
	END_VAR
END_FUNCTION_BLOCK
```

#### ScrewLoading.st
```iecst
(* TODO: Add your comment here *)
FUNCTION_BLOCK ScrewLoading

	//---Spustenie
	IF EDGEPOS(Cmd.AutomatStart=1) THEN
		Internal.Step.Brzda:=1;
		Internal.Step.VibracnyHrniec:=1;
	ELSIF EDGEPOS (Cmd.ManualStartHrniec) THEN
		Internal.Step.VibracnyHrniec:=120;
	ELSIF EDGEPOS (Cmd.ManualPresunBrzdu) THEN
		Internal.Step.Brzda:=120;
	ELSIF EDGEPOS(Cmd.AutomatStart=0) OR EDGEPOS(Cmd.ManualStartHrniec=0) THEN
		Internal.Step.Brzda:=0;
		Internal.Step.VibracnyHrniec:=140;
	END_IF

	//Mapovanie ovladania
	IN.Brzda.VyziadanieSkrutky:=Cmd.PodajSkrutku;
	Status.SkrutkaPripravena:=OUT.Brzda.SktutkaPodana;

	//Run signal
	IF Internal.Step.VibracnyHrniec>120 AND Cmd.ManualStartHrniec=1 THEN
		Status.AutomatBezi:=0;
		Status.ManualBeziHrniec:=1;
	ELSIF Internal.Step.VibracnyHrniec>=100 AND Cmd.AutomatStart=1 THEN
		Status.AutomatBezi:=1;
		Status.ManualBeziHrniec:=0;
	ELSIF Internal.Step.VibracnyHrniec=0 THEN
		Status.AutomatBezi:=0;
		Status.ManualBeziHrniec:=0;
	END_IF

	//---Ovladanie brzdy--------------------------------------------------------------
	CASE Internal.Step.Brzda OF
		//---Vypnute-------------------
		0: Internal.Status.Brzda:="Vypnute";
			OUT.Brzda.NastrelenieSkrutky:=0;
			OUT.Brzda.OdsavanieNecistot:=0;
			OUT.Brzda.PodajSkrutku:=0;
			OUT.Brzda.ZakladnaPoloha:=0;
			OUT.Brzda.SktutkaPodana:=0;

			Internal.Brzda.T_CasCisteniaSkrutky.IN:=0;
			Internal.Brzda.T_PreletSkrutky.IN:=0;
			Internal.Brzda.T_PresunBrzdy.IN:=0;

			//---Inicializacia-------------
		1: Internal.Status.Brzda:="Inicializacia - Kontrolujem polohu brzdy";
			OUT.Brzda.ZakladnaPoloha:=1;
			OUT.Brzda.PodajSkrutku:=0;
			Internal.Brzda.T_PresunBrzdy.IN:=1;

			IF IN.Brzda.PodajSkrutku=0 AND IN.Brzda.ZakladnaPoloha=1 THEN
				Internal.Brzda.T_PresunBrzdy.IN:=0;
				Internal.Step.Brzda:=Internal.Step.Brzda+1;
			ELSIF Internal.Brzda.T_PresunBrzdy.Q=1 THEN
				OUT.Brzda.ZakladnaPoloha:=0;
				OUT.Brzda.PodajSkrutku:=0;
				Internal.Brzda.T_PresunBrzdy.IN:=0;
				Internal.Step.Brzda:=150; // brzda sa neda presunut
			END_IF

		2: Internal.Status.Brzda:="Inicializacia - Kontrolujem pritomnost skrutky";
			IF IN.Brzda.ZakladnaPoloha=1 AND IN.Brzda.SkrutkaPritomnaVBrzde=0 THEN
				Internal.Step.Brzda:=100;
			ELSIF IN.Brzda.ZakladnaPoloha=1 AND IN.Brzda.SkrutkaPritomnaVBrzde=1 THEN
				Internal.Step.Brzda:=102;
			END_IF

			//---Automat-------------
		100: Internal.Status.Brzda:="Automat - Cakam na skrutku";
			IF IN.Brzda.ZakladnaPoloha=1 AND IN.Brzda.SkrutkaPritomnaVBrzde=1 THEN
				Internal.Step.Brzda:=Internal.Step.Brzda+1;
			END_IF

		101: Internal.Status.Brzda:="Automat - Cistim skrutku";
			OUT.Brzda.OdsavanieNecistot:=1;
			Internal.Brzda.T_CasCisteniaSkrutky.IN:=1;

			IF Internal.Brzda.T_CasCisteniaSkrutky.Q=1 THEN
				OUT.Brzda.OdsavanieNecistot:=0;
				Internal.Brzda.T_CasCisteniaSkrutky.IN:=0;
				Internal.Step.Brzda:=Internal.Step.Brzda+1;
			END_IF

		102: Internal.Status.Brzda:="Automat - Cakam na vyziadanie skrutky";
			IF IN.Brzda.VyziadanieSkrutky=1 THEN
				OUT.Brzda.ZakladnaPoloha:=0;
				OUT.Brzda.PodajSkrutku:=1;
				Internal.Brzda.T_PresunBrzdy.IN:=1;
			END_IF

			IF IN.Brzda.PodajSkrutku=1 AND IN.Brzda.ZakladnaPoloha=0 THEN
				OUT.Brzda.OdsavanieNecistot:=1;
				Internal.Brzda.T_PresunBrzdy.IN:=0;
				Internal.Brzda.T_PreletSkrutky.IN:=1;
				OUT.Brzda.NastrelenieSkrutky:=1;
				Internal.Step.Brzda:=Internal.Step.Brzda+1;
			ELSIF Internal.Brzda.T_PresunBrzdy.Q=1 THEN
				OUT.Brzda.ZakladnaPoloha:=0;
				OUT.Brzda.PodajSkrutku:=0;
				Internal.Brzda.T_PresunBrzdy.IN:=0;
				Internal.Step.Brzda:=150; // Brzda sa neda presunut
			END_IF

		103: Internal.Status.Brzda:="Automat - Cakam na prelet skrutky";
			IF IN.Brzda.PreletSkrutky=1 THEN
				OUT.Brzda.NastrelenieSkrutky:=0;
				OUT.Brzda.ZakladnaPoloha:=1;
				OUT.Brzda.PodajSkrutku:=0;
				Internal.Brzda.T_PreletSkrutky.IN:=0;
			ELSIF Internal.Brzda.T_PreletSkrutky.Q=1 THEN
				OUT.Brzda.NastrelenieSkrutky:=0;
				OUT.Brzda.ZakladnaPoloha:=0;
				OUT.Brzda.PodajSkrutku:=0;
				Internal.Brzda.T_PreletSkrutky.IN:=0;
				Internal.Step.Brzda:=151; // Skrutka nepreletela snimacom
			END_IF

			IF IN.Brzda.PodajSkrutku=0 AND IN.Brzda.ZakladnaPoloha=1 THEN
				Internal.Step.Brzda:=Internal.Step.Brzda+1;
			END_IF

		104: Internal.Status.Brzda:="Automat - Skrutka podana";
			OUT.Brzda.SktutkaPodana:=1;

			IF IN.Brzda.VyziadanieSkrutky=0 THEN
				OUT.Brzda.SktutkaPodana:=0;
				Internal.Step.Brzda:=Internal.Step.Brzda+1;
			END_IF

		105: Internal.Status.Brzda:="Automat - Ukoncenie";
			Internal.Step.Brzda:=100;

		120: Internal.Status.Brzda:="Manual - Presuvam brzdu na vypustenie skrutky";

			OUT.Brzda.ZakladnaPoloha:=0;
			OUT.Brzda.PodajSkrutku:= 1;

			IF Cmd.ManualPresunBrzdu=0 THEN
				OUT.Brzda.PodajSkrutku:= 0;
				OUT.Brzda.ZakladnaPoloha:=1;
				IF IN.Brzda.ZakladnaPoloha THEN
					Internal.Step.Brzda:=0;
				END_IF
			END_IF

			//---Error-----------------------
		150: Internal.Status.Brzda:="Error - Brzda sa neda presunut";
			Error.ErrorBit:=1;
			Error.ErrorNumber:=1;
			Error.ErrorMessage:=Internal.Status.Brzda;
		151: Internal.Status.Brzda:="Error - Skrutka nepresla preletovym snimacom";
			Error.ErrorBit:=1;
			Error.ErrorNumber:=2;
			Error.ErrorMessage:=Internal.Status.Brzda;

			//---Manual----------------------
		250: Internal.Status.Brzda:="Manual - Presuvam brzdu";
			OUT.Brzda.PodajSkrutku:=1;
			OUT.Brzda.ZakladnaPoloha:=0;

			IF Cmd.ManualPresunBrzdu=0 THEN
				OUT.Brzda.PodajSkrutku:=0;
				OUT.Brzda.ZakladnaPoloha:=1;
				Internal.Step.Brzda:=0;
			END_IF
	END_CASE

	//---Ovladanie vibracneho hrnca-------------------------------------------------------------
	CASE Internal.Step.VibracnyHrniec OF
		//---Vypnute-------------------
		0: Internal.Status.VibracnyHrniec:="Vypnute";

			OUT.VibracnyHrniec.VzduchNastreleniaSkrutky:=0;
			OUT.VibracnyHrniec.OddelovacVysunut:=0;
			OUT.VibracnyHrniec.PrerusenieZasobovaniaSkrutiek:=0;
			OUT.VibracnyHrniec.TiedenieSkrutiek:=0;
			OUT.VibracnyHrniec.ZapniVibromotor:=0;

			Internal.VibracnyHrniec.T_PreletSkrutky.IN:=0;
			Internal.VibracnyHrniec.T_ZapnutieTriediacehoVzduchu.IN:=0;
			Internal.VibracnyHrniec.T_Zaplnenie.IN:=0;
			Internal.VibracnyHrniec.T_PredOpatovnymPodanimSkrutky.IN:=0;

			Error.ErrorBit:=0;
			Error.ErrorNumber:=0;
			Error.ErrorMessage:="";

			//---Inicializacia-------------
		1: Internal.Status.VibracnyHrniec:="Inicializacia - Zapinam vibracny hrniec";
			OUT.VibracnyHrniec.TiedenieSkrutiek:=1;
			Internal.VibracnyHrniec.T_ZapnutieTriediacehoVzduchu.IN:=1;

			IF Internal.VibracnyHrniec.T_ZapnutieTriediacehoVzduchu.Q=1 THEN
				Internal.VibracnyHrniec.T_ZapnutieTriediacehoVzduchu.IN:=0;
				OUT.VibracnyHrniec.ZapniVibromotor:=1;
				Internal.Step.VibracnyHrniec:=100;
			END_IF

			//---Automat-------------------
		100: Internal.Status.VibracnyHrniec:="Automat - Cakam na uvolnenie brzdy";
			IF IN.VibracnyHrniec.VibracnaListaZaplnena=1 THEN
				Internal.VibracnyHrniec.T_Zaplnenie.IN:=1;
			ELSE
				Internal.VibracnyHrniec.T_Zaplnenie.IN:=0;
			END_IF

			IF IN.VibracnyHrniec.VibracnaListaZaplnena=1 AND Internal.VibracnyHrniec.T_Zaplnenie.Q=1 AND (Internal.Step.Brzda=102 OR Internal.Step.Brzda=104) THEN
				Internal.VibracnyHrniec.T_Zaplnenie.IN:=0;
				Internal.Step.VibracnyHrniec:=105;
			ELSIF Internal.Step.Brzda=100 AND OUT.VibracnyHrniec.ZapniVibromotor=0 THEN
				Internal.VibracnyHrniec.T_Zaplnenie.IN:=0;
				Internal.Step.VibracnyHrniec:=110;
			ELSIF Internal.Step.Brzda=100 AND OUT.VibracnyHrniec.ZapniVibromotor=1 THEN
				Internal.VibracnyHrniec.T_Zaplnenie.IN:=0;
				Internal.Step.VibracnyHrniec:=111;
			END_IF

			//---Vypnutie hrnca po čase z fázy 100
		105: Internal.Status.VibracnyHrniec:="Automat - Vypinam hrniec";
			OUT.VibracnyHrniec.ZapniVibromotor:=0;
			Internal.VibracnyHrniec.T_ZapnutieTriediacehoVzduchu.IN:=1;

			IF Internal.VibracnyHrniec.T_ZapnutieTriediacehoVzduchu.Q=1 THEN
				Internal.VibracnyHrniec.T_ZapnutieTriediacehoVzduchu.IN:=0;
				OUT.VibracnyHrniec.TiedenieSkrutiek:=0;
				Internal.Step.VibracnyHrniec:=100;
			END_IF

			//---Zapnutie hrnca z fázy 100
		110: Internal.Status.VibracnyHrniec:="Automat - Zapinam hrniec";
			OUT.VibracnyHrniec.TiedenieSkrutiek:=1;
			Internal.VibracnyHrniec.T_ZapnutieTriediacehoVzduchu.IN:=1;

			IF Internal.VibracnyHrniec.T_ZapnutieTriediacehoVzduchu.Q=1 THEN
				Internal.VibracnyHrniec.T_ZapnutieTriediacehoVzduchu.IN:=0;
				OUT.VibracnyHrniec.ZapniVibromotor:=1;
				Internal.Step.VibracnyHrniec:=Internal.Step.VibracnyHrniec+1;
			END_IF

		111: Internal.Status.VibracnyHrniec:="Automat - Podavam skrutku";
			IF IN.VibracnyHrniec.VibracnaListaZaplnena=1 THEN
				Internal.VibracnyHrniec.T_Zaplnenie.IN:=1;
			ELSE
				Internal.VibracnyHrniec.T_Zaplnenie.IN:=0;
			END_IF

			IF Internal.VibracnyHrniec.T_Zaplnenie.Q=1 THEN
				OUT.VibracnyHrniec.OddelovacVysunut:=1;
				Internal.VibracnyHrniec.T_PreletSkrutky.IN:=1;
			END_IF

			IF IN.VibracnyHrniec.PreletovySnimac=1 THEN
				Internal.VibracnyHrniec.T_PreletSkrutky.IN:=0;
				Internal.VibracnyHrniec.T_Zaplnenie.IN:=0;
				Internal.Step.VibracnyHrniec:=114;
			ELSIF Internal.VibracnyHrniec.T_PreletSkrutky.Q=1 THEN
				OUT.VibracnyHrniec.OddelovacVysunut:=0;
				Internal.VibracnyHrniec.T_Zaplnenie.IN:=0;
				Internal.VibracnyHrniec.T_PreletSkrutky.IN:=0;
				Internal.Step.VibracnyHrniec:=112;// Skrutka sa neda podat
			END_IF

		112: Internal.Status.VibracnyHrniec:="Automat - Cakam na opatovne podanie skrutky";

			Internal.VibracnyHrniec.T_PredOpatovnymPodanimSkrutky.IN:=1;

			IF Internal.VibracnyHrniec.T_PredOpatovnymPodanimSkrutky.Q THEN
				Internal.VibracnyHrniec.T_PredOpatovnymPodanimSkrutky.IN:=0;
				Internal.Step.VibracnyHrniec:=111;
			END_IF

		114: Internal.Status.VibracnyHrniec:="Automat - Nastrelovanie";
			OUT.VibracnyHrniec.OddelovacVysunut:=0;
			OUT.VibracnyHrniec.VzduchNastreleniaSkrutky:=1;

			IF Internal.Step.Brzda>100 THEN
				OUT.VibracnyHrniec.VzduchNastreleniaSkrutky:=0;
				Internal.Step.VibracnyHrniec:=Internal.Step.VibracnyHrniec+1;
			END_IF

		115: Internal.Status.VibracnyHrniec:="Automat - Koniec cyklu";
			Internal.Step.VibracnyHrniec:=100;

			//---Manualne vibrovanie
		120: Internal.Status.VibracnyHrniec:="Manual - Zapinam vibracny hrniec";
			OUT.VibracnyHrniec.TiedenieSkrutiek:=1;
			Internal.VibracnyHrniec.T_ZapnutieTriediacehoVzduchu.IN:=1;

			IF Internal.VibracnyHrniec.T_ZapnutieTriediacehoVzduchu.Q=1 THEN
				Internal.VibracnyHrniec.T_ZapnutieTriediacehoVzduchu.IN:=0;
				OUT.VibracnyHrniec.ZapniVibromotor:=1;
				Internal.Step.VibracnyHrniec:=121;
			END_IF

			//---Automat-------------------
		121: Internal.Status.VibracnyHrniec:="Manual - Prebieha vynasanie skrutiek";
			IF IN.VibracnyHrniec.VibracnaListaZaplnena=1 THEN
				Internal.VibracnyHrniec.T_Zaplnenie.IN:=1;
			ELSE
				Internal.VibracnyHrniec.T_Zaplnenie.IN:=0;
			END_IF

			IF IN.VibracnyHrniec.VibracnaListaZaplnena=1 AND Internal.VibracnyHrniec.T_Zaplnenie.Q=1 AND OUT.VibracnyHrniec.ZapniVibromotor THEN
				OUT.VibracnyHrniec.PrerusenieZasobovaniaSkrutiek:=1;
			ELSE
				OUT.VibracnyHrniec.PrerusenieZasobovaniaSkrutiek:=0;
			END_IF

			//---Ukoncenie vibrovania
		140: Internal.Status.VibracnyHrniec:="Ukoncenie - Vypinam vibracny hrniec";
			OUT.VibracnyHrniec.ZapniVibromotor:=0;
			Internal.VibracnyHrniec.T_ZapnutieTriediacehoVzduchu.IN:=1;

			IF Internal.VibracnyHrniec.T_ZapnutieTriediacehoVzduchu.Q=1 THEN
				Internal.VibracnyHrniec.T_ZapnutieTriediacehoVzduchu.IN:=0;
				OUT.VibracnyHrniec.TiedenieSkrutiek:=0;
				Internal.Step.VibracnyHrniec:=0;
			END_IF

			//---Error-----------------------
		150: Internal.Status.VibracnyHrniec:="Error - Skrutka sa neda podat";
			Error.ErrorBit:=1;
			Error.ErrorNumber:=3;
			Error.ErrorMessage:=Internal.Status.VibracnyHrniec;
			OUT.VibracnyHrniec.TiedenieSkrutiek:=0;
			OUT.VibracnyHrniec.ZapniVibromotor:=0;

			//---Manual----------------------
		250: Internal.Status.VibracnyHrniec:="Manual";
	END_CASE

	IF IN.VibracnyHrniec.VibracnaListaZaplnena=1 AND Internal.Step.VibracnyHrniec>99 AND OUT.VibracnyHrniec.ZapniVibromotor THEN
		OUT.VibracnyHrniec.PrerusenieZasobovaniaSkrutiek:=1;
	ELSE
		OUT.VibracnyHrniec.PrerusenieZasobovaniaSkrutiek:=0;
	END_IF

	//---Casovace-------------------------------------------------------------------------------
	Internal.Brzda.T_CasCisteniaSkrutky.PT:=T#1s;//REAL_TO_TIME(Visu.Premenne.);
	Internal.Brzda.T_CasCisteniaSkrutky();

	Internal.Brzda.T_PreletSkrutky.PT:=T#5s;//REAL_TO_TIME(Visu.Premenne.);
	Internal.Brzda.T_PreletSkrutky();

	Internal.Brzda.T_PresunBrzdy.PT:=T#2s;//REAL_TO_TIME(Visu.Premenne.);
	Internal.Brzda.T_PresunBrzdy();

	Internal.VibracnyHrniec.T_PreletSkrutky.PT:=T#5s;//REAL_TO_TIME(Visu.Premenne.);
	Internal.VibracnyHrniec.T_PreletSkrutky();

	Internal.VibracnyHrniec.T_ZapnutieTriediacehoVzduchu.PT:=T#0.5s;//REAL_TO_TIME(Visu.Premenne.);
	Internal.VibracnyHrniec.T_ZapnutieTriediacehoVzduchu();

	Internal.VibracnyHrniec.T_Zaplnenie.PT:=T#1s;//REAL_TO_TIME(Visu.Premenne.);
	Internal.VibracnyHrniec.T_Zaplnenie();

	Internal.VibracnyHrniec.T_PredOpatovnymPodanimSkrutky.PT:=T#2s;//REAL_TO_TIME(Visu.Premenne.);
	Internal.VibracnyHrniec.T_PredOpatovnymPodanimSkrutky();

END_FUNCTION_BLOCK
```

### Library Logical/Libraries/SKTcp (ANSIC, version 1.00.9) - Panasonic TCP Client Traceabilita
Depends on: AsBrStr, AsTCP, sys_lib, standard, IecCheck, FileIO

#### Types.typ - Exported data types
```iecst
(*

         projekt: SKTcp - Panasonic

         autor: Ing. Milan Jun
         company: B+R Automatizace spol. s r.o.
         date: 10.09.2020

*)

TYPE
	SKTcpClientSC_Type : 	STRUCT
		StepName : STRING[255];
		bNext : BOOL;
		bJump : BOOL;
		bLast : BOOL;
		bRepeat : BOOL;
		edge : BOOL;
		step : UINT;
		idle_time : TON;
		alarm_time : TON;
	END_STRUCT;
END_TYPE

(**)

TYPE
	SKTcpClientTraceStatus_Type : 	STRUCT
		RecvSize : UDINT;
		DataRecv : ARRAY[0..MAX_STRING_MINUS_ONE]OF USINT;
		RecvCounter : UDINT;
		enaSend : BOOL;
		staReceived : BOOL;
		staSent : BOOL;
		staError : BOOL;
		staErrorSent : BOOL;
		staErrorOpen : BOOL;
		staErrorRecv : BOOL;
		staErrorIoctl : BOOL;
		staErrorClose : BOOL;
		staErrorClient : BOOL;
		staErrorRecvTout : BOOL;
		staErrorConn : BOOL;
		staErrorConnTout : BOOL;
		staSending : BOOL;
		staReceiving : BOOL;
		staReadyToClose : BOOL;
		staReadyToSend : BOOL;
	END_STRUCT;
	SKTcpClientTraceParPackInter_Typ : 	STRUCT
		start : USINT;
		length_b_int : UINT;
		length_int : UINT;
		length_str : STRING[5];
		xor : BYTE;
		xor_str : USINT;
		stop : USINT;
		ti : USINT;
		length : UINT;
		ret_len : UINT;
	END_STRUCT;
	SKTcpClientTraceParams_Type : 	STRUCT
		IPaddrServ : ARRAY[0..39]OF USINT;
		IPportClient : UINT;
		IPportServ : UINT;
		disRecv : BOOL;
		enaClose : BOOL; (*Zatvorenie portu po prijati odpovede od servera*)
		RecvTimeout : UDINT := 5000;
		ConnTimeout : UDINT := 5000;
		Packet : SKTcpClientTraceParamsPack_Typ;
	END_STRUCT;
	SKTcpClientTraceParamsPack_Typ : 	STRUCT
		internal : SKTcpClientTraceParPackInter_Typ;
		type : STRING[1];
		workplace : STRING[5];
		rfid : STRING[10];
		master : STRING[30];
		dps1 : STRING[30];
		dps2 : STRING[30];
		dps3 : STRING[30];
		dps4 : STRING[30];
		dps5 : STRING[30];
		operator_id : STRING[8];
		data_report : STRING[MAX_STRING];
		result : STRING[4];
	END_STRUCT;
	SKTcpClientTraceLogger_Typ : 	STRUCT
		empty : USINT;
	END_STRUCT;
	SKTcpClientTraceIntern_Type : 	STRUCT
		Step : UINT;
		TCP_Open : TcpOpen;
		TCP_Close : TcpClose;
		TCP_Client : TcpClient;
		TCP_Recv : TcpRecv;
		TCP_Send : TcpSend;
		TCP_Ioctl : TcpIoctl;
		linger_opt : tcpLINGER_typ;
		TimerRecv : TON;
		TimerConn : TON;
		TimerIddle : TON;
		cmdClose : BOOL;
		cmdSend : BOOL;
		CloseOld : BOOL;
		SendOld : BOOL;
		EnableOld : BOOL;
		Splitter : SKTcpClientSplitter;
		oneskorenie : TON;
		SKTcpLogger : SKTcpLogger;
	END_STRUCT;
	SKTcpClientTraceDataSend_Type : 	STRUCT
		send_data_a : ARRAY[0..MAX_STRING_MINUS_ONE]OF USINT;
		send_data_b : ARRAY[0..MAX_STRING_MINUS_ONE]OF USINT;
		DataSend : ARRAY[0..MAX_STRING_MINUS_ONE]OF USINT;
	END_STRUCT;
	SKTcpClientTraceCmd_Type : 	STRUCT
		Send : BOOL;
		Close : BOOL;
		LoggerOn : BOOL;
	END_STRUCT;
	SKTcpClientTestParPackInter_Type : 	STRUCT
		start : USINT;
		data_length : UINT;
		length : USINT;
		xor : USINT;
		stop : USINT;
		ti : USINT;
	END_STRUCT;
END_TYPE

(**)

TYPE
	SKTcpClientTesterStatus_Type : 	STRUCT
		RecvSize : UDINT;
		DataRecv : ARRAY[0..199]OF USINT;
		RecvCounter : UDINT;
		enaSend : BOOL;
		staReceived : BOOL;
		staSent : BOOL;
		staError : BOOL;
		staErrorSent : BOOL;
		staErrorOpen : BOOL;
		staErrorRecv : BOOL;
		staErrorIoctl : BOOL;
		staErrorClose : BOOL;
		staErrorClient : BOOL;
		staErrorRecvTout : BOOL;
		staErrorConn : BOOL;
		staErrorConnTout : BOOL;
		staSending : BOOL;
		staReceiving : BOOL;
		staReadyToClose : BOOL;
		staReadyToSend : BOOL;
	END_STRUCT;
	SKTcpClientTesterParams_Type : 	STRUCT
		IPaddrServ : ARRAY[0..39]OF USINT;
		IPportClient : UINT;
		IPportServ : UINT;
		disRecv : BOOL;
		enaClose : BOOL; (*Zatvorenie portu po prijati odpovede od servera*)
		RecvTimeout : UDINT := 3000;
		ConnTimeout : UDINT := 3000;
		Packet : SKTcpClientTesterParamsPack_Type;
	END_STRUCT;
	SKTcpClientTesterParamsPack_Type : 	STRUCT
		type : USINT;
		workplace : USINT;
		id : USINT;
		data : ARRAY[0..31]OF USINT;
		internal : SKTcpClientTestParPackInter_Type;
	END_STRUCT;
	SKTcpClientTesterLogger_Typ : 	STRUCT
		empty : USINT;
	END_STRUCT;
	SKTcpClientTesterIntern_Type : 	STRUCT
		Step : UINT;
		Ident : UDINT;
		TCP_Open : TcpOpen;
		TCP_Close : TcpClose;
		TCP_Client : TcpClient;
		TCP_Recv : TcpRecv;
		TCP_Send : TcpSend;
		TCP_Ioctl : TcpIoctl;
		linger_opt : tcpLINGER_typ;
		TimerRecv : TON;
		TimerConn : TON;
		cmdClose : BOOL;
		cmdSend : BOOL;
		CloseOld : BOOL;
		SendOld : BOOL;
		EnableOld : BOOL;
	END_STRUCT;
	SKTcpClientTesterDataSend_Type : 	STRUCT
		SendLength : UDINT;
		send_data_a : ARRAY[0..199]OF USINT;
		DataSend : ARRAY[0..199]OF USINT;
	END_STRUCT;
	SKTcpClientTesterCmd_Type : 	STRUCT
		Send : BOOL;
		Close : BOOL;
	END_STRUCT;
END_TYPE

(**)

TYPE
	SKTcpLoggerInternal_Typ : 	STRUCT
		step : USINT;
		data : STRING[MAX_STRING];
		FileOpen : FileOpen;
		FileClose : FileClose;
		FileWrite : FileWrite;
	END_STRUCT;
END_TYPE
```

#### Constants.var - Exported constants
```iecst
(*

         projekt: SKTcp - Panasonic

         autor: Ing. Milan Jun
         company: B+R Automatizace spol. s r.o.
         date: 10.09.2020

*)
VAR CONSTANT
	MAX_CHARACTER : UINT := 1;
	MAX_STRING : UINT := 5000;
	MAX_STRING_MINUS_ONE : UINT := 4999;
END_VAR
```

#### SKTcp.fun - Exported functions and function blocks
```iecst
(**************************************************************

         projekt: SKTcp - Panasonic

         autor: Ing. Milan Jun
         company: B+R Automatizace spol. s r.o.
         date: 10.09.2020

*)

{REDUND_ERROR} FUNCTION_BLOCK SKTcpClientSplitter (*SKTcpClient - Splitter*) (*$GROUP=User,$CAT=User,$GROUPICON=User.png,$CATICON=User.png*)
	VAR_INPUT
		enable : BOOL;
		iSelector : USINT;
		iInputString : STRING[MAX_STRING];
	END_VAR
	VAR_OUTPUT
		out : ARRAY[0..14] OF STRING[MAX_STRING];
		done : BOOL;
		OUT_Master : STRING[30];
		OUT_Typ : STRING[1];
		OUT_Result : STRING[2];
	END_VAR
	VAR
		enableOld : BOOL;
		tmpInputString : ARRAY[0..MAX_STRING_MINUS_ONE] OF USINT;
		tmpString : STRING[MAX_CHARACTER];
		idx : ARRAY[0..1] OF UDINT;
	END_VAR
END_FUNCTION_BLOCK

{REDUND_ERROR} FUNCTION_BLOCK SKTcpClientTester (*SKTcpClient - Tester*) (*$GROUP=User,$CAT=User,$GROUPICON=User.png,$CATICON=User.png*)
	VAR_INPUT
		Enable : BOOL;
		Cmd : SKTcpClientTesterCmd_Type;
		Params : SKTcpClientTesterParams_Type;
		DataSend : SKTcpClientTesterDataSend_Type;
	END_VAR
	VAR_OUTPUT
		Status : SKTcpClientTesterStatus_Type;
		FBStatus : {REDUND_UNREPLICABLE} UINT;
		logger : SKTcpClientTesterLogger_Typ;
	END_VAR
	VAR
		Internal : SKTcpClientTesterIntern_Type;
	END_VAR
END_FUNCTION_BLOCK

{REDUND_ERROR} FUNCTION_BLOCK SKTcpClientTrace (*SKTcpClient - ZberDat verzia 2*) (*$GROUP=User,$CAT=User,$GROUPICON=User.png,$CATICON=User.png*)
	VAR_INPUT
		Enable : BOOL;
		Cmd : SKTcpClientTraceCmd_Type;
		Params : SKTcpClientTraceParams_Type;
		DataSend : SKTcpClientTraceDataSend_Type;
		pDevice : UDINT;
		pFile : UDINT;
	END_VAR
	VAR_OUTPUT
		Status : SKTcpClientTraceStatus_Type;
		FBStatus : {REDUND_UNREPLICABLE} UINT;
		logger : SKTcpClientTraceLogger_Typ;
	END_VAR
	VAR
		Internal : SKTcpClientTraceIntern_Type;
	END_VAR
END_FUNCTION_BLOCK

{REDUND_ERROR} FUNCTION_BLOCK SKTcpClientEdge (*SKTcpClient - Edge*) (*$GROUP=User,$CAT=User,$GROUPICON=User.png,$CATICON=User.png*)
	VAR_INPUT
		CLK : BOOL;
	END_VAR
	VAR_OUTPUT
		Q : {REDUND_UNREPLICABLE} BOOL;
	END_VAR
	VAR
		Last_State : BOOL;
	END_VAR
END_FUNCTION_BLOCK

{REDUND_ERROR} FUNCTION_BLOCK SKTcpLogger (*SKTcpLogger*) (*$GROUP=User,$CAT=User,$GROUPICON=User.png,$CATICON=User.png*)
	VAR_INPUT
		enable : BOOL;
		trigger : BOOL;
		pDevice : UDINT;
		pFile : UDINT;
		pSrc : UDINT;
		mode : USINT;
	END_VAR
	VAR_OUTPUT
		active : BOOL;
		done : BOOL;
	END_VAR
	VAR
		internal : SKTcpLoggerInternal_Typ;
	END_VAR
END_FUNCTION_BLOCK

{REDUND_ERROR} FUNCTION SKTcpClientNod : UINT (*SKTcpClient - Number Of Digits*) (*$GROUP=User,$CAT=User,$GROUPICON=User.png,$CATICON=User.png*)
	VAR_INPUT
		n : UDINT;
	END_VAR
END_FUNCTION

{REDUND_ERROR} FUNCTION SKTcpClientXor : USINT (*SKTcpClient - Xor*) (*$GROUP=User,$CAT=User,$GROUPICON=User.png,$CATICON=User.png*)
	VAR_INPUT
		in : ARRAY[0..4999] OF USINT;
		len : UINT;
	END_VAR
END_FUNCTION

{REDUND_ERROR} FUNCTION SKTcpClientNewCsvEntry : USINT (*SKTcpClient - New CSV Entries*) (*$GROUP=User,$CAT=User,$GROUPICON=User.png,$CATICON=User.png*)
	VAR_INPUT
		IDstep : STRING[10];
		Description : STRING[100];
		TypeValue : STRING[10];
		MinTol : STRING[10];
		MaxTol : STRING[10];
		Nom : STRING[10];
		MinEle : STRING[10];
		MaxEle : STRING[10];
		Value : STRING[10];
		ValEle : STRING[10];
		Result : STRING[10];
		pData : UDINT;
	END_VAR
END_FUNCTION

{REDUND_ERROR} FUNCTION SKTcpClientNewLoggerEntry : USINT (*SKTcpClient - New Logger Entries*)
	VAR_INPUT
		msg : STRING[1100];
		pData : UDINT;
		entrys : UINT;
	END_VAR
END_FUNCTION

{REDUND_ERROR} FUNCTION SKTcpClientSC : USINT (*SKTcpClient - SC*) (*$GROUP=User,$CAT=User,$GROUPICON=User.png,$CATICON=User.png*)
	VAR_INPUT
		sc : SKTcpClientSC_Type;
	END_VAR
END_FUNCTION
```

#### SKTcpClientTester.c - SKTcpClientTester
```c
/*************************************************************
*
*         projekt: SKTcp - Panasonic
*
*         autor: Ing. Milan Jun
*         company: B+R Automatizace spol. s r.o.
*         date: 10.09.2020
*
*/

#include <bur/plctypes.h>
#ifdef __cplusplus
	extern "C"
	{
#endif
#include "SKTcp.h"
#ifdef __cplusplus
	};
#endif

/* SKTcpClientTester */
void SKTcpClientTester(struct SKTcpClientTester* inst)
{

	if( inst->Enable == 1 ) {

		if(( inst->Cmd.Send == 1 ) && ( inst->Internal.SendOld == 0 )) {
			inst->Internal.cmdSend = 1 ;
		}
		inst->Internal.SendOld = inst->Cmd.Send ;

		if(( inst->Cmd.Close == 1 ) && ( inst->Internal.CloseOld == 0 )) {
			inst->Internal.cmdClose = 1 ;
		} else {
			if( inst->Cmd.Close == 0 ) {
				inst->Internal.cmdClose = 0 ;
			}
		}
		inst->Internal.CloseOld = inst->Cmd.Close ;

		inst->Status.staSending = 0 ;
		inst->Status.staReceiving = 0 ;
		inst->Status.staReadyToSend = 0 ;
		inst->Status.staReadyToClose = 0 ;

		switch( inst->Internal.Step ) {

			case 0:
				inst->Status.staReadyToSend = 1 ;

				if( inst->Internal.cmdSend == 1 ) {
					inst->FBStatus = 0xFFFF ;
					inst->Status.staSent = 0 ;
					inst->Status.staReceived = 0 ;

					inst->Status.staError = 0 ;
					inst->Status.staErrorSent = 0 ;
					inst->Status.staErrorOpen = 0 ;
					inst->Status.staErrorRecv = 0 ;
					inst->Status.staErrorRecvTout = 0 ;
					inst->Status.staErrorOpen = 0 ;
					inst->Status.staErrorIoctl = 0 ;
					inst->Status.staErrorClient = 0 ;
					inst->Status.staErrorConn = 0 ;
					inst->Status.staErrorConnTout = 0 ;

					inst->Status.RecvSize = 0 ;
					memset((void*)&inst->Status.DataRecv[0], 0, sizeof(inst->Status.DataRecv)) ;

					inst->Internal.TimerConn.IN = 1 ;
					inst->Internal.TimerConn.PT = inst->Params.ConnTimeout ;

					inst->Internal.TCP_Open.enable = 1;
					inst->Internal.TCP_Open.pIfAddr = 0;
					inst->Internal.TCP_Open.port = inst->Params.IPportClient;
					inst->Internal.TCP_Open.options = 0;
					TcpOpen(&inst->Internal.TCP_Open);

					if( inst->Internal.TCP_Open.status == 0 ) {
						//inst->Internal.cmdSend = 0 ;
						inst->Internal.Ident = inst->Internal.TCP_Open.ident ;
						inst->Internal.Step = 5;
					}
					else if( inst->Internal.TimerConn.Q == 1 ) {
						//      inst->Internal.cmdSend = 0 ;
						inst->Status.staErrorOpen = 1 ;
						inst->Status.staErrorConn = 1 ;
						inst->Status.staErrorConnTout = 1 ;
						inst->Internal.Step = 99;
					} else if( inst->Internal.TCP_Open.status == ERR_FUB_BUSY ) {

					} else {
						if( inst->Internal.TCP_Open.status == tcpERR_ALREADY_EXIST ) {
							inst->Status.staErrorOpen = 1 ;
							inst->Internal.Step = 90;
						} else {
							inst->Status.staErrorOpen = 1 ;
							inst->Internal.Step = 99;
						}
						//inst->Internal.cmdSend = 0 ;
					}
				}

				    else if( inst->Cmd.Close == 1 ) {
				     inst->Cmd.Close = 0 ;
				     inst->Internal.Step = 40 ;
				    }
				break ;

			case 5:
				inst->Internal.linger_opt.lLinger = 0;
				inst->Internal.linger_opt.lOnOff = 1;

				inst->Internal.TCP_Ioctl.enable = 1;
				inst->Internal.TCP_Ioctl.ident = inst->Internal.Ident;
				inst->Internal.TCP_Ioctl.ioctl = tcpSO_LINGER_SET;
				inst->Internal.TCP_Ioctl.pData = (UDINT)&(inst->Internal.linger_opt);
				inst->Internal.TCP_Ioctl.datalen = sizeof(inst->Internal.linger_opt);
				TcpIoctl(&inst->Internal.TCP_Ioctl);

				if( inst->Internal.TCP_Ioctl.status == 0 ) {
					inst->Internal.Step = 10;
				} else if( inst->Internal.TimerConn.Q == 1 ) {
					inst->Status.staErrorOpen = 1 ;
					inst->Status.staErrorConn = 1 ;
					inst->Status.staErrorConnTout = 1 ;
					inst->Internal.Step = 99;
				} else if( inst->Internal.TCP_Ioctl.status == ERR_FUB_BUSY ) {
				} else {
					inst->Status.staErrorIoctl = 1 ;
					inst->Internal.Step = 90;
				}
				break ;

			case 10:
				inst->Internal.TCP_Client.enable = 1;
				inst->Internal.TCP_Client.ident = inst->Internal.Ident ;
				inst->Internal.TCP_Client.portserv = inst->Params.IPportServ ;
				inst->Internal.TCP_Client.pServer = (UDINT)&inst->Params.IPaddrServ[0];
				TcpClient(&inst->Internal.TCP_Client) ;

				if( inst->Internal.TCP_Client.status == 0 ) {
					inst->Internal.Step = 15;
				} else if( inst->Internal.TimerConn.Q == 1 ) {
					inst->Status.staErrorOpen = 1 ;
					inst->Status.staErrorConn = 1 ;
					inst->Status.staErrorConnTout = 1 ;
					inst->Internal.Step = 90;
				} else if( inst->Internal.TCP_Client.status == ERR_FUB_BUSY ) {
				} else if( inst->Internal.TCP_Client.status == tcpERR_INVALID ) {
					inst->Status.staErrorClient = 1 ;
					inst->Status.staErrorConn = 1 ;
					inst->Internal.Step = 90;
				} else {
					inst->Status.staErrorClient = 1 ;
					inst->Internal.Step = 90;
				}
				break ;

			case 15:
				inst->Status.staReadyToSend = 1 ;
				inst->Status.staReadyToClose = 1 ;
				inst->Status.staSending = 0 ;

				if( inst->Cmd.Send == 1 ) {
					inst->Status.RecvSize = 0 ;
					inst->Internal.TimerRecv.IN = 0 ;
					memset((void*)&inst->Status.DataRecv[0], 0, sizeof(inst->Status.DataRecv)) ;
					inst->Internal.Step = 19;
				} else if( inst->Internal.cmdClose == 1 ) {
					inst->Internal.cmdClose = 0 ;
					inst->Internal.Step = 40;
				}
				break ;

			case 19:

				inst->Params.Packet.internal.start = 2;
				inst->Params.Packet.internal.xor = 0;
				inst->Params.Packet.internal.stop = 3;

				if ( inst->Params.Packet.type == 0 || inst->Params.Packet.type == 2 || inst->Params.Packet.type == 3 )
					inst->Params.Packet.internal.length = 3;
				else if ( inst->Params.Packet.type == 1 )
					inst->Params.Packet.internal.length = 34;

				inst->Params.Packet.internal.data_length = inst->Params.Packet.internal.length + SKTcpClientNod(inst->Params.Packet.internal.length);

				memset((UDINT)&(inst->DataSend.send_data_a), 0, sizeof(inst->DataSend.send_data_a));

				inst->DataSend.send_data_a[0] = inst->Params.Packet.internal.data_length;
				inst->DataSend.send_data_a[1] = inst->Params.Packet.type;
				inst->DataSend.send_data_a[2] = inst->Params.Packet.workplace;
				inst->DataSend.send_data_a[3] = inst->Params.Packet.id;

				if (  inst->Params.Packet.type == 1  ) {

					for (inst->Params.Packet.internal.ti = 0; inst->Params.Packet.internal.ti < 32; inst->Params.Packet.internal.ti++)
					{
						inst->DataSend.send_data_a[inst->Params.Packet.internal.ti+4] = inst->Params.Packet.data[inst->Params.Packet.internal.ti];
					}
				}

				// Vypocet XOR
				for (inst->Params.Packet.internal.ti = 0; inst->Params.Packet.internal.ti < inst->Params.Packet.internal.data_length; inst->Params.Packet.internal.ti++)
				{
					inst->Params.Packet.internal.xor = inst->Params.Packet.internal.xor ^ inst->DataSend.send_data_a[inst->Params.Packet.internal.ti];
				}

				memset((UDINT)&(inst->DataSend.DataSend), 0, sizeof(inst->DataSend.DataSend));
				inst->DataSend.DataSend[0] = inst->Params.Packet.internal.start;
				inst->DataSend.DataSend[1] = inst->Params.Packet.internal.data_length;
				inst->DataSend.DataSend[2] = inst->Params.Packet.type;
				inst->DataSend.DataSend[3] = inst->Params.Packet.workplace;
				inst->DataSend.DataSend[4] = inst->Params.Packet.id;
				if (inst->Params.Packet.type == 0 || inst->Params.Packet.type == 2 || inst->Params.Packet.type == 3)
				{
					inst->DataSend.DataSend[5] = inst->Params.Packet.internal.xor;
					inst->DataSend.DataSend[6] = inst->Params.Packet.internal.stop;
				}

				else if (  inst->Params.Packet.type == 1  ) {

					for (inst->Params.Packet.internal.ti = 0; inst->Params.Packet.internal.ti < 32; inst->Params.Packet.internal.ti++)
					{
						inst->DataSend.DataSend[inst->Params.Packet.internal.ti+5] = inst->Params.Packet.data[inst->Params.Packet.internal.ti];

					}
					inst->DataSend.DataSend[37] = inst->Params.Packet.internal.xor;
					inst->DataSend.DataSend[38] = inst->Params.Packet.internal.stop;
				}

				inst->Internal.Step = 20;

				break;

			case 20:

				inst->Status.staSending = 1 ;
				inst->Status.staSent = 0 ;

				inst->Internal.TCP_Send.enable = 1;
				inst->Internal.TCP_Send.ident = inst->Internal.Ident;
				inst->Internal.TCP_Send.pData = (UDINT)&inst->DataSend.DataSend;

				if ( inst->Params.Packet.type == 0 || inst->Params.Packet.type == 2 || inst->Params.Packet.type == 3  )
				{
					inst->Internal.TCP_Send.datalen = inst->Params.Packet.internal.data_length + 3;
				}
				if ( inst->Params.Packet.type == 1  )
				{
					inst->Internal.TCP_Send.datalen = inst->Params.Packet.internal.data_length + 3;
				}

				inst->Internal.TCP_Send.flags = 0;
				TcpSend(&inst->Internal.TCP_Send);

				if( inst->Internal.TCP_Send.status == 0 ) {
					inst->Status.staSent = 1 ;
					if( inst->Params.disRecv == 0 ) {
						inst->Internal.TimerRecv.IN = 0 ;
						inst->Internal.Step = 30;
					}
				} else if( inst->Internal.TCP_Send.status == ERR_FUB_BUSY )	{
				} else if (( inst->Internal.TCP_Send.status == tcpERR_SENTLEN )
				|| ( inst->Internal.TCP_Send.status == tcpERR_NOT_CONNECTED )) {
					inst->Internal.Step = 90;
				} else {
					inst->Status.staErrorSent = 1 ;
					inst->Internal.Step = 90;
				}
				break ;

			case 30:
				inst->Status.staReceiving = 1 ;
				inst->Status.staReceived = 0 ;

				inst->Internal.TimerRecv.IN = 1 ;
				inst->Internal.TimerRecv.PT = inst->Params.RecvTimeout ;

				inst->Internal.TCP_Recv.enable = 1;
				inst->Internal.TCP_Recv.ident = inst->Internal.Ident;
				inst->Internal.TCP_Recv.pData	= (UDINT)&inst->Status.DataRecv[0];
				inst->Internal.TCP_Recv.datamax = sizeof(inst->Status.DataRecv);
				inst->Internal.TCP_Recv.flags = 0;
				TcpRecv(&inst->Internal.TCP_Recv);

				if( inst->Internal.TCP_Recv.status == 0 ) {
					inst->Status.staReceived = 1 ;
					inst->Status.RecvSize = inst->Internal.TCP_Recv.recvlen;
					inst->Status.RecvCounter++ ;

					if( inst->Params.enaClose == 1 ) {
						inst->Internal.Step = 40;
					} else {
						inst->Internal.Step = 15 ;
					}
				} else if( inst->Internal.TCP_Recv.status == tcpERR_NO_DATA ) {
					if( inst->Internal.TimerRecv.Q == 1 ) {
						inst->Status.staErrorRecvTout = 1 ;
						inst->Internal.Step = 90;
					}
				} else if( inst->Internal.TCP_Recv.status == ERR_FUB_BUSY ) {
					if( inst->Internal.TimerRecv.Q == 1 ) {

					}
				} else if( inst->Internal.TCP_Recv.status == tcpERR_NOT_CONNECTED ) {
					inst->Status.staErrorRecv = 1 ;
					inst->Internal.Step = 90;
				} else if( inst->Internal.TimerRecv.Q == 1 ) {
					inst->Status.staErrorRecv = 1 ;
					inst->Internal.TimerRecv.IN = 0 ;
					inst->Internal.Step = 90;
				}
				break ;

			case 40:
				inst->Internal.TCP_Close.enable = 1;
				inst->Internal.TCP_Close.ident = inst->Internal.Ident ;
				inst->Internal.TCP_Close.how = 0;
				TcpClose(&inst->Internal.TCP_Close);

				if( inst->Internal.TCP_Close.status == 0 ) {
					inst->Internal.Ident = 0 ;
					inst->Internal.Step = 100;
					inst->Status.staReceived = 1 ;
				} else if( inst->Internal.TCP_Close.status == ERR_FUB_BUSY ) {
				} else {
					inst->Status.staErrorClose = 1 ;
					inst->Internal.Step = 99;
				}
				break ;

			case 90:
				inst->Internal.TCP_Close.enable = 1;
				inst->Internal.TCP_Close.ident = inst->Internal.Ident;
				inst->Internal.TCP_Close.how = 0;
				TcpClose(&inst->Internal.TCP_Close);

				if( inst->Internal.TCP_Close.status == 0 ) {
					inst->Internal.Ident = 0 ;
					inst->Internal.Step = 99;
				} else if( inst->Internal.TCP_Close.status == ERR_FUB_BUSY ) {
				} else {
					inst->Status.staErrorClose = 1 ;
					inst->Internal.Step = 99;
				}
				break ;

			case 99:
				inst->FBStatus = 1 ;
				inst->Status.staError = 1 ; ;
				inst->Internal.Step = 0;
				inst->Internal.TimerConn.IN = 0 ;
				inst->Internal.cmdSend = 0 ;
				break ;

			case 100:
				inst->FBStatus = 0 ;
				inst->Internal.Step = 0;
				inst->Internal.cmdSend = 0 ;
				inst->Internal.TimerConn.IN = 0 ;
				break ;

		}
	} else {
		if( inst->Cmd.Send == 0 ) {
			inst->FBStatus = 0xFFFE ;
		}

		if( inst->Internal.Ident != 0 ) {
			inst->Internal.TCP_Close.enable = 1;
			inst->Internal.TCP_Close.ident = inst->Internal.Ident;
			inst->Internal.TCP_Close.how = 0;
			TcpClose(&inst->Internal.TCP_Close);

			if( inst->Internal.TCP_Close.status == 0 ) {
				inst->Internal.Ident = 0 ;
			} else if( inst->Internal.TCP_Close.status == ERR_FUB_BUSY ) {
			} else {
			}
		}
		inst->Internal.TimerRecv.IN = 0 ;
		inst->Internal.TimerConn.IN = 0 ;
		inst->Internal.Step = 0 ;
	}

	inst->Internal.EnableOld = inst->Enable ;
	TON(&inst->Internal.TimerRecv) ;
	TON(&inst->Internal.TimerConn) ;

}
```
